LIN {X 0,Y 682.192,Z 1116.485,A -85,B 0,C 180,E1 25132.947,E2 25132.947} C_VEL
LIN {X 0,Y 681.497,Z 1132.896,A -85,B 0,C 180,E1 25130.835,E2 25130.835} C_VEL
LIN {X 0,Y 681.036,Z 1145.573,A -85,B 0,C 180,E1 25129,E2 25129} C_VEL
LIN {X 0,Y 680.643,Z 1157.899,A -85,B 0,C 180,E1 25126.991,E2 25126.991} C_VEL
LIN {X 0,Y 680.337,Z 1169.837,A -85,B 0,C 180,E1 25124.73,E2 25124.73} C_VEL
LIN {X 0,Y 680.158,Z 1178.436,A -85,B 0,C 180,E1 25122.826,E2 25122.826} C_VEL
LIN {X 0,Y 680.019,Z 1186.222,A -85,B 0,C 180,E1 25120.82,E2 25120.82} C_VEL
LIN {X 0,Y 679.964,Z 1193.353,A -85,B 0,C 180,E1 25118.541,E2 25118.541} C_VEL
LIN {X 0,Y 679.927,Z 1198.829,A -85,B 0,C 180,E1 25116.216,E2 25116.216} C_VEL
LIN {X 0,Y 679.913,Z 1202.374,A -85,B 0,C 180,E1 25114.048,E2 25114.048} C_VEL
LIN {X 0,Y 679.907,Z 1204.493,A -85,B 0,C 180,E1 25111.77,E2 25111.77} C_VEL
LIN {X 0,Y 679.891,Z 1204.872,A -85,B 0,C 180,E1 25109.495,E2 25109.495} C_VEL
LIN {X 0,Y 679.907,Z 1203.956,A -85,B 0,C 180,E1 25107.472,E2 25107.472} C_VEL
LIN {X 0,Y 679.912,Z 1201.428,A -85,B 0,C 180,E1 25105.276,E2 25105.276} C_VEL
LIN {X 0,Y 679.934,Z 1197.152,A -85,B 0,C 180,E1 25102.99,E2 25102.99} C_VEL
LIN {X 0,Y 679.978,Z 1191.385,A -85,B 0,C 180,E1 25100.777,E2 25100.777} C_VEL
LIN {X 0,Y 680.067,Z 1184.278,A -85,B 0,C 180,E1 25098.638,E2 25098.638} C_VEL
LIN {X 0,Y 680.24,Z 1173.938,A -85,B 0,C 180,E1 25096.138,E2 25096.138} C_VEL
LIN {X 0,Y 680.464,Z 1164.538,A -85,B 0,C 180,E1 25094.227,E2 25094.227} C_VEL
LIN {X 0,Y 680.75,Z 1154.23,A -85,B 0,C 180,E1 25092.388,E2 25092.388} C_VEL
LIN {X 0,Y 681.149,Z 1141.939,A -85,B 0,C 180,E1 25090.447,E2 25090.447} C_VEL
LIN {X 0,Y 681.795,Z 1125.467,A -85,B 0,C 180,E1 25088.177,E2 25088.177} C_VEL
LIN {X 0,Y 682.441,Z 1111.072,A -85,B 0,C 180,E1 25086.423,E2 25086.423} C_VEL
LIN {X 0,Y 683.271,Z 1093.72,A -85,B 0,C 180,E1 25084.518,E2 25084.518} C_VEL
LIN {X 0,Y 684.267,Z 1074.728,A -85,B 0,C 180,E1 25082.679,E2 25082.679} C_VEL
LIN {X 0,Y 685.157,Z 1057.951,A -85,B 0,C 180,E1 25081.212,E2 25081.212} C_VEL
LIN {X 0,Y 686.261,Z 1038.591,A -85,B 0,C 180,E1 25079.679,E2 25079.679} C_VEL
LIN {X 0,Y 687.621,Z 1015.177,A -85,B 0,C 180,E1 25078.043,E2 25078.043} C_VEL
LIN {X 0,Y 688.735,Z 995.445,A -85,B 0,C 180,E1 25076.818,E2 25076.818} C_VEL
LIN {X 0,Y 689.844,Z 975.494,A -85,B 0,C 180,E1 25075.709,E2 25075.709} C_VEL
LIN {X 0,Y 691.118,Z 951.69,A -85,B 0,C 180,E1 25074.54,E2 25074.54} C_VEL
LIN {X 0,Y 692.335,Z 926.424,A -85,B 0,C 180,E1 25073.487,E2 25073.487} C_VEL
LIN {X 0,Y 693.317,Z 904.137,A -85,B 0,C 180,E1 25072.695,E2 25072.695} C_VEL
LIN {X 0,Y 694.253,Z 881.059,A -85,B 0,C 180,E1 25072.001,E2 25072.001} C_VEL
LIN {X 0,Y 695.167,Z 854.051,A -85,B 0,C 180,E1 25071.355,E2 25071.355} C_VEL
LIN {X 0,Y 695.825,Z 826.957,A -85,B 0,C 180,E1 25070.881,E2 25070.881} C_VEL
LIN {X 0,Y 698.216,Z 605.17,A -85,B 0,C 180,E1 25068.081,E2 25068.081} C_VEL
LIN {X 0,Y 700.479,Z 401.113,A -85,B 0,C 180,E1 25065.437,E2 25065.437} C_VEL
LIN {X 0,Y 700.65,Z 371.915,A -85,B 0,C 180,E1 25065.038,E2 25065.038} C_VEL
LIN {X 0,Y 697.922,Z 362.234,A -85,B 0,C 180,E1 25064.675,E2 25064.675} C_VEL
LIN {X 0,Y 690.093,Z 350.368,A -85,B 0,C 180,E1 25063.818,E2 25063.818} C_VEL
LIN {X 0,Y 683.619,Z 336.797,A -85,B 0,C 180,E1 25062.172,E2 25062.172} C_VEL
LIN {X 0,Y 681.934,Z 333.218,A -85,B 0,C 180,E1 25061.729,E2 25061.729} C_VEL
LIN {X 0,Y 680.487,Z 329.763,A -85,B 0,C 180,E1 25061.314,E2 25061.314} C_VEL
LIN {X 0,Y 680.455,Z 329.473,A -85,B 0,C 180,E1 25061.171,E2 25061.171} C_VEL
LIN {X 0,Y 680.483,Z 329.469,A -85,B 0,C 180,E1 25058.108,E2 25058.108} C_VEL
LIN {X 0,Y 680.435,Z 329.466,A -85,B 0,C 180,E1 25055.482,E2 25055.482} C_VEL
LIN {X 0,Y 680.45,Z 329.467,A -85,B 0,C 180,E1 25052.936,E2 25052.936} C_VEL
LIN {X 0,Y 680.456,Z 329.462,A -85,B 0,C 180,E1 25049.78,E2 25049.78} C_VEL
LIN {X 0,Y 680.427,Z 329.462,A -85,B 0,C 180,E1 25047.249,E2 25047.249} C_VEL
LIN {X 0,Y 680.448,Z 329.464,A -85,B 0,C 180,E1 25044.666,E2 25044.666} C_VEL
LIN {X 0,Y 680.443,Z 329.453,A -85,B 0,C 180,E1 25041.542,E2 25041.542} C_VEL
LIN {X 0,Y 680.419,Z 329.47,A -85,B 0,C 180,E1 25039.04,E2 25039.04} C_VEL
LIN {X 0,Y 680.439,Z 329.451,A -85,B 0,C 180,E1 25036.476,E2 25036.476} C_VEL
LIN {X 0,Y 680.438,Z 329.466,A -85,B 0,C 180,E1 25033.339,E2 25033.339} C_VEL
LIN {X 0,Y 680.416,Z 329.454,A -85,B 0,C 180,E1 25030.842,E2 25030.842} C_VEL
LIN {X 0,Y 680.444,Z 329.47,A -85,B 0,C 180,E1 25028.28,E2 25028.28} C_VEL
LIN {X 0,Y 680.446,Z 329.459,A -85,B 0,C 180,E1 25025.143,E2 25025.143} C_VEL
LIN {X 0,Y 680.427,Z 329.468,A -85,B 0,C 180,E1 25022.611,E2 25022.611} C_VEL
LIN {X 0,Y 680.462,Z 329.448,A -85,B 0,C 180,E1 25020,E2 25020} C_VEL
LIN {X 0,Y 680.449,Z 329.464,A -85,B 0,C 180,E1 25016.883,E2 25016.883} C_VEL
LIN {X 0,Y 680.432,Z 329.449,A -85,B 0,C 180,E1 25014.35,E2 25014.35} C_VEL
LIN {X 0,Y 680.495,Z 329.469,A -85,B 0,C 180,E1 25011.636,E2 25011.636} C_VEL
LIN {X 0,Y 680.452,Z 329.458,A -85,B 0,C 180,E1 25008.644,E2 25008.644} C_VEL
LIN {X 0,Y 680.443,Z 329.466,A -85,B 0,C 180,E1 25006.141,E2 25006.141} C_VEL
LIN {X 0,Y 680.523,Z 329.45,A -85,B 0,C 180,E1 25003.263,E2 25003.263} C_VEL
LIN {X 0,Y 680.452,Z 329.455,A -85,B 0,C 180,E1 25000.336,E2 25000.336} C_VEL
LIN {X 0,Y 680.457,Z 329.465,A -85,B 0,C 180,E1 24997.778,E2 24997.778} C_VEL
LIN {X 0,Y 680.518,Z 329.449,A -85,B 0,C 180,E1 24994.78,E2 24994.78} C_VEL
LIN {X 0,Y 680.455,Z 329.464,A -85,B 0,C 180,E1 24991.951,E2 24991.951} C_VEL
LIN {X 0,Y 680.471,Z 329.465,A -85,B 0,C 180,E1 24989.482,E2 24989.482} C_VEL
LIN {X 0,Y 679.538,Z 329.59,A -85,B 0,C 180,E1 24988.834,E2 24988.834} C_VEL
LIN {X 0,Y 673.042,Z 330.4,A -85,B 0,C 180,E1 24986.969,E2 24986.969} C_VEL
LIN {X 0,Y 672.579,Z 330.454,A -85,B 0,C 180,E1 24986.544,E2 24986.544} C_VEL
LIN {X 0,Y 672.608,Z 330.615,A -85,B 0,C 180,E1 24984.551,E2 24984.551} C_VEL
LIN {X 0,Y 673.956,Z 334.1,A -85,B 0,C 180,E1 24984.124,E2 24984.124} C_VEL
LIN {X 0,Y 677.383,Z 341.291,A -85,B 0,C 180,E1 24983.233,E2 24983.233} C_VEL
LIN {X 0,Y 692.08,Z 362.695,A -85,B 0,C 180,E1 24981.619,E2 24981.619} C_VEL
LIN {X 0,Y 695.109,Z 367.708,A -85,B 0,C 180,E1 24981.292,E2 24981.292} C_VEL
LIN {X 0,Y 692.375,Z 585.7,A -85,B 0,C 180,E1 24978.44,E2 24978.44} C_VEL
LIN {X 0,Y 689.696,Z 812.863,A -85,B 0,C 180,E1 24975.554,E2 24975.554} C_VEL
LIN {X 0,Y 689.06,Z 837.442,A -85,B 0,C 180,E1 24975.148,E2 24975.148} C_VEL
LIN {X 0,Y 688.188,Z 863.617,A -85,B 0,C 180,E1 24974.567,E2 24974.567} C_VEL
LIN {X 0,Y 687.053,Z 889.758,A -85,B 0,C 180,E1 24973.816,E2 24973.816} C_VEL
LIN {X 0,Y 686.051,Z 911.255,A -85,B 0,C 180,E1 24973.069,E2 24973.069} C_VEL
LIN {X 0,Y 685.026,Z 930.752,A -85,B 0,C 180,E1 24972.289,E2 24972.289} C_VEL
LIN {X 0,Y 683.925,Z 950.165,A -85,B 0,C 180,E1 24971.409,E2 24971.409} C_VEL
LIN {X 0,Y 682.742,Z 969.945,A -85,B 0,C 180,E1 24970.398,E2 24970.398} C_VEL
LIN {X 0,Y 681.349,Z 992.918,A -85,B 0,C 180,E1 24969.075,E2 24969.075} C_VEL
LIN {X 0,Y 679.821,Z 1015.891,A -85,B 0,C 180,E1 24967.555,E2 24967.555} C_VEL
LIN {X 0,Y 678.685,Z 1034.023,A -85,B 0,C 180,E1 24966.211,E2 24966.211} C_VEL
LIN {X 0,Y 677.553,Z 1052.755,A -85,B 0,C 180,E1 24964.677,E2 24964.677} C_VEL
LIN {X 0,Y 676.24,Z 1074.005,A -85,B 0,C 180,E1 24962.719,E2 24962.719} C_VEL
LIN {X 0,Y 675.312,Z 1090.747,A -85,B 0,C 180,E1 24960.986,E2 24960.986} C_VEL
LIN {X 0,Y 674.385,Z 1108.733,A -85,B 0,C 180,E1 24958.904,E2 24958.904} C_VEL
LIN {X 0,Y 673.661,Z 1123.806,A -85,B 0,C 180,E1 24956.916,E2 24956.916} C_VEL
LIN {X 0,Y 673.147,Z 1136.6,A -85,B 0,C 180,E1 24955.029,E2 24955.029} C_VEL
LIN {X 0,Y 672.653,Z 1150.249,A -85,B 0,C 180,E1 24952.735,E2 24952.735} C_VEL
LIN {X 0,Y 672.371,Z 1160.899,A -85,B 0,C 180,E1 24950.636,E2 24950.636} C_VEL
LIN {X 0,Y 672.18,Z 1169.232,A -85,B 0,C 180,E1 24948.741,E2 24948.741} C_VEL
LIN {X 0,Y 672.043,Z 1176.964,A -85,B 0,C 180,E1 24946.687,E2 24946.687} C_VEL
LIN {X 0,Y 671.967,Z 1183.913,A -85,B 0,C 180,E1 24944.388,E2 24944.388} C_VEL
LIN {X 0,Y 671.924,Z 1189.086,A -85,B 0,C 180,E1 24942.111,E2 24942.111} C_VEL
LIN {X 0,Y 671.91,Z 1192.514,A -85,B 0,C 180,E1 24939.94,E2 24939.94} C_VEL
LIN {X 0,Y 671.907,Z 1194.57,A -85,B 0,C 180,E1 24937.61,E2 24937.61} C_VEL
LIN {X 0,Y 671.898,Z 1194.855,A -85,B 0,C 180,E1 24935.379,E2 24935.379} C_VEL
LIN {X 0,Y 671.907,Z 1193.966,A -85,B 0,C 180,E1 24933.412,E2 24933.412} C_VEL
LIN {X 0,Y 671.914,Z 1191.456,A -85,B 0,C 180,E1 24931.193,E2 24931.193} C_VEL
LIN {X 0,Y 671.941,Z 1187.221,A -85,B 0,C 180,E1 24928.891,E2 24928.891} C_VEL
LIN {X 0,Y 671.989,Z 1181.533,A -85,B 0,C 180,E1 24926.673,E2 24926.673} C_VEL
LIN {X 0,Y 672.093,Z 1174.22,A -85,B 0,C 180,E1 24924.44,E2 24924.44} C_VEL
LIN {X 0,Y 672.267,Z 1164.112,A -85,B 0,C 180,E1 24921.963,E2 24921.963} C_VEL
LIN {X 0,Y 672.539,Z 1154.496,A -85,B 0,C 180,E1 24919.982,E2 24919.982} C_VEL
LIN {X 0,Y 672.864,Z 1144.443,A -85,B 0,C 180,E1 24918.166,E2 24918.166} C_VEL
LIN {X 0,Y 673.321,Z 1131.955,A -85,B 0,C 180,E1 24916.167,E2 24916.167} C_VEL
LIN {X 0,Y 674.037,Z 1115.678,A -85,B 0,C 180,E1 24913.895,E2 24913.895} C_VEL
LIN {X 0,Y 674.762,Z 1100.696,A -85,B 0,C 180,E1 24912.048,E2 24912.048} C_VEL
LIN {X 0,Y 675.765,Z 1083.129,A -85,B 0,C 180,E1 24910.104,E2 24910.104} C_VEL
LIN {X 0,Y 676.829,Z 1063.955,A -85,B 0,C 180,E1 24908.235,E2 24908.235} C_VEL
LIN {X 0,Y 677.883,Z 1046.646,A -85,B 0,C 180,E1 24906.715,E2 24906.715} C_VEL
LIN {X 0,Y 679.31,Z 1025.059,A -85,B 0,C 180,E1 24905.011,E2 24905.011} C_VEL
LIN {X 0,Y 680.632,Z 1003.591,A -85,B 0,C 180,E1 24903.522,E2 24903.522} C_VEL
LIN {X 0,Y 681.817,Z 984.728,A -85,B 0,C 180,E1 24902.347,E2 24902.347} C_VEL
LIN {X 0,Y 683.115,Z 963.487,A -85,B 0,C 180,E1 24901.165,E2 24901.165} C_VEL
LIN {X 0,Y 684.679,Z 937.06,A -85,B 0,C 180,E1 24899.892,E2 24899.892} C_VEL
LIN {X 0,Y 685.803,Z 915.856,A -85,B 0,C 180,E1 24899.015,E2 24899.015} C_VEL
LIN {X 0,Y 686.762,Z 895.765,A -85,B 0,C 180,E1 24898.292,E2 24898.292} C_VEL
LIN {X 0,Y 687.782,Z 873.499,A -85,B 0,C 180,E1 24897.609,E2 24897.609} C_VEL
LIN {X 0,Y 688.802,Z 846.613,A -85,B 0,C 180,E1 24896.945,E2 24896.945} C_VEL
LIN {X 0,Y 689.546,Z 819.591,A -85,B 0,C 180,E1 24896.454,E2 24896.454} C_VEL
LIN {X 0,Y 690.716,Z 728.303,A -85,B 0,C 180,E1 24895.287,E2 24895.287} C_VEL
LIN {X 0,Y 693.173,Z 517.537,A -85,B 0,C 180,E1 24892.586,E2 24892.586} C_VEL
LIN {X 0,Y 695.013,Z 367.196,A -85,B 0,C 180,E1 24890.603,E2 24890.603} C_VEL
LIN {X 0,Y 681.213,Z 346.68,A -85,B 0,C 180,E1 24889.106,E2 24889.106} C_VEL
LIN {X 0,Y 676.997,Z 340.608,A -85,B 0,C 180,E1 24888.616,E2 24888.616} C_VEL
LIN {X 0,Y 673.889,Z 333.927,A -85,B 0,C 180,E1 24887.766,E2 24887.766} C_VEL
LIN {X 0,Y 672.576,Z 330.451,A -85,B 0,C 180,E1 24887.319,E2 24887.319} C_VEL
LIN {X 0,Y 672.555,Z 330.455,A -85,B 0,C 180,E1 24884.349,E2 24884.349} C_VEL
LIN {X 0,Y 672.579,Z 330.449,A -85,B 0,C 180,E1 24881.345,E2 24881.345} C_VEL
LIN {X 0,Y 672.555,Z 330.453,A -85,B 0,C 180,E1 24878.419,E2 24878.419} C_VEL
LIN {X 0,Y 672.585,Z 330.446,A -85,B 0,C 180,E1 24875.436,E2 24875.436} C_VEL
LIN {X 0,Y 672.552,Z 330.456,A -85,B 0,C 180,E1 24872.359,E2 24872.359} C_VEL
LIN {X 0,Y 672.579,Z 330.447,A -85,B 0,C 180,E1 24869.38,E2 24869.38} C_VEL
LIN {X 0,Y 672.548,Z 330.431,A -85,B 0,C 180,E1 24866.298,E2 24866.298} C_VEL
LIN {X 0,Y 672.559,Z 330.449,A -85,B 0,C 180,E1 24863.388,E2 24863.388} C_VEL
LIN {X 0,Y 672.549,Z 330.429,A -85,B 0,C 180,E1 24860.264,E2 24860.264} C_VEL
LIN {X 0,Y 672.536,Z 330.451,A -85,B 0,C 180,E1 24857.477,E2 24857.477} C_VEL
LIN {X 0,Y 672.572,Z 330.425,A -85,B 0,C 180,E1 24854.375,E2 24854.375} C_VEL
LIN {X 0,Y 672.522,Z 330.45,A -85,B 0,C 180,E1 24851.543,E2 24851.543} C_VEL
LIN {X 0,Y 672.588,Z 330.446,A -85,B 0,C 180,E1 24848.636,E2 24848.636} C_VEL
LIN {X 0,Y 672.518,Z 330.449,A -85,B 0,C 180,E1 24845.717,E2 24845.717} C_VEL
LIN {X 0,Y 672.525,Z 330.453,A -85,B 0,C 180,E1 24843.068,E2 24843.068} C_VEL
LIN {X 0,Y 672.541,Z 330.456,A -85,B 0,C 180,E1 24839.915,E2 24839.915} C_VEL
LIN {X 0,Y 672.504,Z 330.453,A -85,B 0,C 180,E1 24837.273,E2 24837.273} C_VEL
LIN {X 0,Y 672.564,Z 330.448,A -85,B 0,C 180,E1 24834.455,E2 24834.455} C_VEL
LIN {X 0,Y 672.503,Z 330.451,A -85,B 0,C 180,E1 24831.449,E2 24831.449} C_VEL
LIN {X 0,Y 672.498,Z 330.456,A -85,B 0,C 180,E1 24828.901,E2 24828.901} C_VEL
LIN {X 0,Y 672.576,Z 330.427,A -85,B 0,C 180,E1 24825.976,E2 24825.976} C_VEL
LIN {X 0,Y 672.488,Z 330.458,A -85,B 0,C 180,E1 24823.146,E2 24823.146} C_VEL
LIN {X 0,Y 672.49,Z 330.439,A -85,B 0,C 180,E1 24820.636,E2 24820.636} C_VEL
LIN {X 0,Y 672.539,Z 330.458,A -85,B 0,C 180,E1 24817.629,E2 24817.629} C_VEL
LIN {X 0,Y 672.477,Z 330.434,A -85,B 0,C 180,E1 24814.89,E2 24814.89} C_VEL
LIN {X 0,Y 672.507,Z 330.458,A -85,B 0,C 180,E1 24812.266,E2 24812.266} C_VEL
LIN {X 0,Y 672.508,Z 330.453,A -85,B 0,C 180,E1 24809.139,E2 24809.139} C_VEL
LIN {X 0,Y 672.491,Z 330.46,A -85,B 0,C 180,E1 24806.624,E2 24806.624} C_VEL
LIN {X 0,Y 672.537,Z 330.459,A -85,B 0,C 180,E1 24803.931,E2 24803.931} C_VEL
LIN {X 0,Y 672.515,Z 330.464,A -85,B 0,C 180,E1 24800.905,E2 24800.905} C_VEL
LIN {X 0,Y 672.607,Z 330.647,A -85,B 0,C 180,E1 24799.373,E2 24799.373} C_VEL
LIN {X 0,Y 673.722,Z 333.767,A -85,B 0,C 180,E1 24799.005,E2 24799.005} C_VEL
LIN {X 0,Y 674.749,Z 335.752,A -85,B 0,C 180,E1 24798.743,E2 24798.743} C_VEL
LIN {X 0,Y 680.465,Z 347.723,A -85,B 0,C 180,E1 24797.244,E2 24797.244} C_VEL
LIN {X 0,Y 682.244,Z 351.282,A -85,B 0,C 180,E1 24796.838,E2 24796.838} C_VEL
LIN {X 0,Y 693.378,Z 368.095,A -85,B 0,C 180,E1 24795.621,E2 24795.621} C_VEL
LIN {X 0,Y 695.107,Z 375.541,A -85,B 0,C 180,E1 24795.368,E2 24795.368} C_VEL
LIN {X 0,Y 692.464,Z 587.805,A -85,B 0,C 180,E1 24792.587,E2 24792.587} C_VEL
LIN {X 0,Y 689.907,Z 810.343,A -85,B 0,C 180,E1 24789.763,E2 24789.763} C_VEL
LIN {X 0,Y 689.271,Z 840.613,A -85,B 0,C 180,E1 24789.32,E2 24789.32} C_VEL
LIN {X 0,Y 688.468,Z 865.299,A -85,B 0,C 180,E1 24788.812,E2 24788.812} C_VEL
LIN {X 0,Y 687.48,Z 890.926,A -85,B 0,C 180,E1 24788.136,E2 24788.136} C_VEL
LIN {X 0,Y 686.225,Z 918.026,A -85,B 0,C 180,E1 24787.235,E2 24787.235} C_VEL
LIN {X 0,Y 685.097,Z 939.47,A -85,B 0,C 180,E1 24786.39,E2 24786.39} C_VEL
LIN {X 0,Y 683.956,Z 959.707,A -85,B 0,C 180,E1 24785.477,E2 24785.477} C_VEL
LIN {X 0,Y 682.726,Z 980.321,A -85,B 0,C 180,E1 24784.424,E2 24784.424} C_VEL
LIN {X 0,Y 681.2,Z 1004.925,A -85,B 0,C 180,E1 24782.995,E2 24782.995} C_VEL
LIN {X 0,Y 679.764,Z 1026.908,A -85,B 0,C 180,E1 24781.528,E2 24781.528} C_VEL
LIN {X 0,Y 678.598,Z 1045.712,A -85,B 0,C 180,E1 24780.125,E2 24780.125} C_VEL
LIN {X 0,Y 677.318,Z 1066.768,A -85,B 0,C 180,E1 24778.376,E2 24778.376} C_VEL
LIN {X 0,Y 676.139,Z 1085.449,A -85,B 0,C 180,E1 24776.621,E2 24776.621} C_VEL
LIN {X 0,Y 675.284,Z 1101.386,A -85,B 0,C 180,E1 24774.961,E2 24774.961} C_VEL
LIN {X 0,Y 674.296,Z 1120.132,A -85,B 0,C 180,E1 24772.77,E2 24772.77} C_VEL
LIN {X 0,Y 673.636,Z 1134.458,A -85,B 0,C 180,E1 24770.869,E2 24770.869} C_VEL
LIN {X 0,Y 673.123,Z 1147.165,A -85,B 0,C 180,E1 24768.985,E2 24768.985} C_VEL
LIN {X 0,Y 672.64,Z 1160.81,A -85,B 0,C 180,E1 24766.672,E2 24766.672} C_VEL
LIN {X 0,Y 672.363,Z 1171.07,A -85,B 0,C 180,E1 24764.644,E2 24764.644} C_VEL
LIN {X 0,Y 672.177,Z 1179.152,A -85,B 0,C 180,E1 24762.806,E2 24762.806} C_VEL
LIN {X 0,Y 672.03,Z 1186.718,A -85,B 0,C 180,E1 24760.805,E2 24760.805} C_VEL
LIN {X 0,Y 671.969,Z 1193.594,A -85,B 0,C 180,E1 24758.558,E2 24758.558} C_VEL
LIN {X 0,Y 671.929,Z 1198.936,A -85,B 0,C 180,E1 24756.237,E2 24756.237} C_VEL
LIN {X 0,Y 671.915,Z 1202.371,A -85,B 0,C 180,E1 24754.096,E2 24754.096} C_VEL
LIN {X 0,Y 671.907,Z 1204.494,A -85,B 0,C 180,E1 24751.791,E2 24751.791} C_VEL
LIN {X 0,Y 671.891,Z 1204.872,A -85,B 0,C 180,E1 24749.489,E2 24749.489} C_VEL
LIN {X 0,Y 671.907,Z 1203.953,A -85,B 0,C 180,E1 24747.442,E2 24747.442} C_VEL
LIN {X 0,Y 671.914,Z 1201.428,A -85,B 0,C 180,E1 24745.22,E2 24745.22} C_VEL
LIN {X 0,Y 671.941,Z 1197.152,A -85,B 0,C 180,E1 24742.906,E2 24742.906} C_VEL
LIN {X 0,Y 671.991,Z 1191.382,A -85,B 0,C 180,E1 24740.667,E2 24740.667} C_VEL
LIN {X 0,Y 672.091,Z 1184.278,A -85,B 0,C 180,E1 24738.501,E2 24738.501} C_VEL
LIN {X 0,Y 672.286,Z 1173.937,A -85,B 0,C 180,E1 24735.971,E2 24735.971} C_VEL
LIN {X 0,Y 672.534,Z 1164.54,A -85,B 0,C 180,E1 24734.036,E2 24734.036} C_VEL
LIN {X 0,Y 672.866,Z 1154.232,A -85,B 0,C 180,E1 24732.175,E2 24732.175} C_VEL
LIN {X 0,Y 673.319,Z 1141.941,A -85,B 0,C 180,E1 24730.21,E2 24730.21} C_VEL
LIN {X 0,Y 674.025,Z 1125.809,A -85,B 0,C 180,E1 24727.957,E2 24727.957} C_VEL
LIN {X 0,Y 674.751,Z 1111.073,A -85,B 0,C 180,E1 24726.138,E2 24726.138} C_VEL
LIN {X 0,Y 675.713,Z 1093.721,A -85,B 0,C 180,E1 24724.212,E2 24724.212} C_VEL
LIN {X 0,Y 676.818,Z 1074.326,A -85,B 0,C 180,E1 24722.315,E2 24722.315} C_VEL
LIN {X 0,Y 677.817,Z 1057.658,A -85,B 0,C 180,E1 24720.845,E2 24720.845} C_VEL
LIN {X 0,Y 679.09,Z 1037.98,A -85,B 0,C 180,E1 24719.276,E2 24719.276} C_VEL
LIN {X 0,Y 680.589,Z 1014.452,A -85,B 0,C 180,E1 24717.623,E2 24717.623} C_VEL
LIN {X 0,Y 681.824,Z 994.646,A -85,B 0,C 180,E1 24716.387,E2 24716.387} C_VEL
LIN {X 0,Y 683.131,Z 973.165,A -85,B 0,C 180,E1 24715.192,E2 24715.192} C_VEL
LIN {X 0,Y 684.732,Z 946.223,A -85,B 0,C 180,E1 24713.9,E2 24713.9} C_VEL
LIN {X 0,Y 685.855,Z 925.015,A -85,B 0,C 180,E1 24713.027,E2 24713.027} C_VEL
LIN {X 0,Y 686.853,Z 904.064,A -85,B 0,C 180,E1 24712.28,E2 24712.28} C_VEL
LIN {X 0,Y 687.876,Z 880.997,A -85,B 0,C 180,E1 24711.584,E2 24711.584} C_VEL
LIN {X 0,Y 688.888,Z 854.053,A -85,B 0,C 180,E1 24710.936,E2 24710.936} C_VEL
LIN {X 0,Y 689.604,Z 827.138,A -85,B 0,C 180,E1 24710.463,E2 24710.463} C_VEL
LIN {X 0,Y 692.229,Z 607.714,A -85,B 0,C 180,E1 24707.669,E2 24707.669} C_VEL
LIN {X 0,Y 694.743,Z 403.368,A -85,B 0,C 180,E1 24705.001,E2 24705.001} C_VEL
LIN {X 0,Y 694.947,Z 374.179,A -85,B 0,C 180,E1 24704.599,E2 24704.599} C_VEL
LIN {X 0,Y 692.936,Z 367.154,A -85,B 0,C 180,E1 24704.328,E2 24704.328} C_VEL
LIN {X 0,Y 683.819,Z 353.781,A -85,B 0,C 180,E1 24703.34,E2 24703.34} C_VEL
LIN {X 0,Y 681.644,Z 350.368,A -85,B 0,C 180,E1 24703.073,E2 24703.073} C_VEL
LIN {X 0,Y 676.08,Z 338.51,A -85,B 0,C 180,E1 24701.61,E2 24701.61} C_VEL
LIN {X 0,Y 673.717,Z 333.758,A -85,B 0,C 180,E1 24700.995,E2 24700.995} C_VEL
LIN {X 0,Y 672.584,Z 330.454,A -85,B 0,C 180,E1 24700.598,E2 24700.598} C_VEL
LIN {X 0,Y 672.504,Z 330.459,A -85,B 0,C 180,E1 24697.668,E2 24697.668} C_VEL
LIN {X 0,Y 672.503,Z 330.454,A -85,B 0,C 180,E1 24695.128,E2 24695.128} C_VEL
LIN {X 0,Y 672.566,Z 330.451,A -85,B 0,C 180,E1 24692.157,E2 24692.157} C_VEL
LIN {X 0,Y 672.493,Z 330.456,A -85,B 0,C 180,E1 24689.384,E2 24689.384} C_VEL
LIN {X 0,Y 672.492,Z 330.449,A -85,B 0,C 180,E1 24686.968,E2 24686.968} C_VEL
LIN {X 0,Y 672.57,Z 330.457,A -85,B 0,C 180,E1 24684.038,E2 24684.038} C_VEL
LIN {X 0,Y 672.485,Z 330.444,A -85,B 0,C 180,E1 24681.272,E2 24681.272} C_VEL
LIN {X 0,Y 672.484,Z 330.459,A -85,B 0,C 180,E1 24678.823,E2 24678.823} C_VEL
LIN {X 0,Y 672.565,Z 330.436,A -85,B 0,C 180,E1 24675.875,E2 24675.875} C_VEL
LIN {X 0,Y 672.481,Z 330.455,A -85,B 0,C 180,E1 24673.062,E2 24673.062} C_VEL
LIN {X 0,Y 672.486,Z 330.442,A -85,B 0,C 180,E1 24670.538,E2 24670.538} C_VEL
LIN {X 0,Y 672.548,Z 330.447,A -85,B 0,C 180,E1 24667.518,E2 24667.518} C_VEL
LIN {X 0,Y 672.486,Z 330.449,A -85,B 0,C 180,E1 24664.776,E2 24664.776} C_VEL
LIN {X 0,Y 672.506,Z 330.458,A -85,B 0,C 180,E1 24662.215,E2 24662.215} C_VEL
LIN {X 0,Y 672.52,Z 330.452,A -85,B 0,C 180,E1 24659.063,E2 24659.063} C_VEL
LIN {X 0,Y 672.494,Z 330.454,A -85,B 0,C 180,E1 24656.42,E2 24656.42} C_VEL
LIN {X 0,Y 672.566,Z 330.439,A -85,B 0,C 180,E1 24653.598,E2 24653.598} C_VEL
LIN {X 0,Y 672.505,Z 330.447,A -85,B 0,C 180,E1 24650.587,E2 24650.587} C_VEL
LIN {X 0,Y 672.511,Z 330.448,A -85,B 0,C 180,E1 24647.986,E2 24647.986} C_VEL
LIN {X 0,Y 672.569,Z 330.43,A -85,B 0,C 180,E1 24645.008,E2 24645.008} C_VEL
LIN {X 0,Y 672.508,Z 330.455,A -85,B 0,C 180,E1 24642.165,E2 24642.165} C_VEL
LIN {X 0,Y 672.562,Z 330.435,A -85,B 0,C 180,E1 24639.369,E2 24639.369} C_VEL
LIN {X 0,Y 672.524,Z 330.448,A -85,B 0,C 180,E1 24636.324,E2 24636.324} C_VEL
LIN {X 0,Y 672.522,Z 330.454,A -85,B 0,C 180,E1 24633.701,E2 24633.701} C_VEL
LIN {X 0,Y 672.588,Z 330.446,A -85,B 0,C 180,E1 24630.718,E2 24630.718} C_VEL
LIN {X 0,Y 672.522,Z 330.456,A -85,B 0,C 180,E1 24627.841,E2 24627.841} C_VEL
LIN {X 0,Y 672.579,Z 330.454,A -85,B 0,C 180,E1 24626.544,E2 24626.544} C_VEL
LIN {X 0,Y 671.671,Z 330.679,A -85,B 0,C 180,E1 24626.089,E2 24626.089} C_VEL
LIN {X 0,Y 668.299,Z 332.282,A -85,B 0,C 180,E1 24625.356,E2 24625.356} C_VEL
LIN {X 0,Y 666.743,Z 334.518,A -85,B 0,C 180,E1 24624.891,E2 24624.891} C_VEL
LIN {X 0,Y 666.809,Z 336.494,A -85,B 0,C 180,E1 24624.619,E2 24624.619} C_VEL
LIN {X 0,Y 669.158,Z 341.54,A -85,B 0,C 180,E1 24623.999,E2 24623.999} C_VEL
LIN {X 0,Y 681.76,Z 359.579,A -85,B 0,C 180,E1 24622.561,E2 24622.561} C_VEL
LIN {X 0,Y 689.425,Z 371.303,A -85,B 0,C 180,E1 24621.719,E2 24621.719} C_VEL
LIN {X 0,Y 686.412,Z 590.021,A -85,B 0,C 180,E1 24618.837,E2 24618.837} C_VEL
LIN {X 0,Y 683.502,Z 813.654,A -85,B 0,C 180,E1 24615.971,E2 24615.971} C_VEL
LIN {X 0,Y 682.82,Z 837.703,A -85,B 0,C 180,E1 24615.57,E2 24615.57} C_VEL
LIN {X 0,Y 681.871,Z 863.883,A -85,B 0,C 180,E1 24614.985,E2 24614.985} C_VEL
LIN {X 0,Y 680.67,Z 889.429,A -85,B 0,C 180,E1 24614.247,E2 24614.247} C_VEL
LIN {X 0,Y 679.567,Z 910.882,A -85,B 0,C 180,E1 24613.499,E2 24613.499} C_VEL
LIN {X 0,Y 678.47,Z 929.901,A -85,B 0,C 180,E1 24612.738,E2 24612.738} C_VEL
LIN {X 0,Y 677.219,Z 950.032,A -85,B 0,C 180,E1 24611.821,E2 24611.821} C_VEL
LIN {X 0,Y 675.915,Z 969.984,A -85,B 0,C 180,E1 24610.794,E2 24610.794} C_VEL
LIN {X 0,Y 674.346,Z 993.619,A -85,B 0,C 180,E1 24609.419,E2 24609.419} C_VEL
LIN {X 0,Y 672.654,Z 1016.598,A -85,B 0,C 180,E1 24607.877,E2 24607.877} C_VEL
LIN {X 0,Y 671.391,Z 1034.83,A -85,B 0,C 180,E1 24606.509,E2 24606.509} C_VEL
LIN {X 0,Y 670.071,Z 1054.857,A -85,B 0,C 180,E1 24604.843,E2 24604.843} C_VEL
LIN {X 0,Y 668.706,Z 1074.695,A -85,B 0,C 180,E1 24602.974,E2 24602.974} C_VEL
LIN {X 0,Y 667.715,Z 1090.61,A -85,B 0,C 180,E1 24601.306,E2 24601.306} C_VEL
LIN {X 0,Y 666.688,Z 1108.577,A -85,B 0,C 180,E1 24599.205,E2 24599.205} C_VEL
LIN {X 0,Y 665.872,Z 1123.898,A -85,B 0,C 180,E1 24597.16,E2 24597.16} C_VEL
LIN {X 0,Y 665.303,Z 1136.579,A -85,B 0,C 180,E1 24595.265,E2 24595.265} C_VEL
LIN {X 0,Y 664.771,Z 1149.955,A -85,B 0,C 180,E1 24592.998,E2 24592.998} C_VEL
LIN {X 0,Y 664.427,Z 1160.963,A -85,B 0,C 180,E1 24590.802,E2 24590.802} C_VEL
LIN {X 0,Y 664.213,Z 1169.289,A -85,B 0,C 180,E1 24588.883,E2 24588.883} C_VEL
LIN {X 0,Y 664.057,Z 1177.011,A -85,B 0,C 180,E1 24586.803,E2 24586.803} C_VEL
LIN {X 0,Y 663.975,Z 1183.982,A -85,B 0,C 180,E1 24584.463,E2 24584.463} C_VEL
LIN {X 0,Y 663.926,Z 1189.11,A -85,B 0,C 180,E1 24582.171,E2 24582.171} C_VEL
LIN {X 0,Y 663.91,Z 1192.563,A -85,B 0,C 180,E1 24579.946,E2 24579.946} C_VEL
LIN {X 0,Y 663.907,Z 1194.573,A -85,B 0,C 180,E1 24577.616,E2 24577.616} C_VEL
LIN {X 0,Y 663.899,Z 1194.851,A -85,B 0,C 180,E1 24575.358,E2 24575.358} C_VEL
LIN {X 0,Y 663.907,Z 1193.952,A -85,B 0,C 180,E1 24573.367,E2 24573.367} C_VEL
LIN {X 0,Y 663.917,Z 1191.435,A -85,B 0,C 180,E1 24571.121,E2 24571.121} C_VEL
LIN {X 0,Y 663.945,Z 1187.189,A -85,B 0,C 180,E1 24568.792,E2 24568.792} C_VEL
LIN {X 0,Y 663.999,Z 1181.49,A -85,B 0,C 180,E1 24566.546,E2 24566.546} C_VEL
LIN {X 0,Y 664.114,Z 1174.211,A -85,B 0,C 180,E1 24564.297,E2 24564.297} C_VEL
LIN {X 0,Y 664.324,Z 1164.051,A -85,B 0,C 180,E1 24561.779,E2 24561.779} C_VEL
LIN {X 0,Y 664.616,Z 1154.432,A -85,B 0,C 180,E1 24559.774,E2 24559.774} C_VEL
LIN {X 0,Y 664.986,Z 1143.865,A -85,B 0,C 180,E1 24557.848,E2 24557.848} C_VEL
LIN {X 0,Y 665.595,Z 1130.176,A -85,B 0,C 180,E1 24555.648,E2 24555.648} C_VEL
LIN {X 0,Y 666.35,Z 1114.779,A -85,B 0,C 180,E1 24553.507,E2 24553.507} C_VEL
LIN {X 0,Y 667.141,Z 1099.849,A -85,B 0,C 180,E1 24551.655,E2 24551.655} C_VEL
LIN {X 0,Y 668.313,Z 1081.252,A -85,B 0,C 180,E1 24549.598,E2 24549.598} C_VEL
LIN {X 0,Y 669.44,Z 1063.177,A -85,B 0,C 180,E1 24547.827,E2 24547.827} C_VEL
LIN {X 0,Y 670.682,Z 1045.42,A -85,B 0,C 180,E1 24546.261,E2 24546.261} C_VEL
LIN {X 0,Y 672.3,Z 1022.368,A -85,B 0,C 180,E1 24544.45,E2 24544.45} C_VEL
LIN {X 0,Y 673.639,Z 1002.717,A -85,B 0,C 180,E1 24543.082,E2 24543.082} C_VEL
LIN {X 0,Y 675.004,Z 982.947,A -85,B 0,C 180,E1 24541.849,E2 24541.849} C_VEL
LIN {X 0,Y 676.732,Z 958.249,A -85,B 0,C 180,E1 24540.49,E2 24540.49} C_VEL
LIN {X 0,Y 678.195,Z 934.629,A -85,B 0,C 180,E1 24539.377,E2 24539.377} C_VEL
LIN {X 0,Y 679.291,Z 915.742,A -85,B 0,C 180,E1 24538.596,E2 24538.596} C_VEL
LIN {X 0,Y 680.347,Z 895.338,A -85,B 0,C 180,E1 24537.858,E2 24537.858} C_VEL
LIN {X 0,Y 681.452,Z 873.122,A -85,B 0,C 180,E1 24537.175,E2 24537.175} C_VEL
LIN {X 0,Y 682.568,Z 846.2,A -85,B 0,C 180,E1 24536.509,E2 24536.509} C_VEL
LIN {X 0,Y 683.37,Z 819.214,A -85,B 0,C 180,E1 24536.02,E2 24536.02} C_VEL
LIN {X 0,Y 684.764,Z 718.371,A -85,B 0,C 180,E1 24534.722,E2 24534.722} C_VEL
LIN {X 0,Y 687.447,Z 510.327,A -85,B 0,C 180,E1 24532.031,E2 24532.031} C_VEL
LIN {X 0,Y 689.298,Z 370.726,A -85,B 0,C 180,E1 24530.172,E2 24530.172} C_VEL
LIN {X 0,Y 673.884,Z 348.149,A -85,B 0,C 180,E1 24528.46,E2 24528.46} C_VEL
LIN {X 0,Y 668.725,Z 340.57,A -85,B 0,C 180,E1 24527.829,E2 24527.829} C_VEL
LIN {X 0,Y 666.082,Z 335.117,A -85,B 0,C 180,E1 24527.102,E2 24527.102} C_VEL
LIN {X 0,Y 664.633,Z 331.51,A -85,B 0,C 180,E1 24526.642,E2 24526.642} C_VEL
LIN {X 0,Y 664.644,Z 331.438,A -85,B 0,C 180,E1 24523.552,E2 24523.552} C_VEL
LIN {X 0,Y 664.621,Z 331.445,A -85,B 0,C 180,E1 24520.536,E2 24520.536} C_VEL
LIN {X 0,Y 664.646,Z 331.434,A -85,B 0,C 180,E1 24517.538,E2 24517.538} C_VEL
LIN {X 0,Y 664.62,Z 331.445,A -85,B 0,C 180,E1 24514.449,E2 24514.449} C_VEL
LIN {X 0,Y 664.64,Z 331.438,A -85,B 0,C 180,E1 24511.462,E2 24511.462} C_VEL
LIN {X 0,Y 664.611,Z 331.435,A -85,B 0,C 180,E1 24508.289,E2 24508.289} C_VEL
LIN {X 0,Y 664.635,Z 331.421,A -85,B 0,C 180,E1 24505.292,E2 24505.292} C_VEL
LIN {X 0,Y 664.604,Z 331.433,A -85,B 0,C 180,E1 24502.187,E2 24502.187} C_VEL
LIN {X 0,Y 664.61,Z 331.42,A -85,B 0,C 180,E1 24499.329,E2 24499.329} C_VEL
LIN {X 0,Y 664.609,Z 331.437,A -85,B 0,C 180,E1 24496.161,E2 24496.161} C_VEL
LIN {X 0,Y 664.588,Z 331.413,A -85,B 0,C 180,E1 24493.397,E2 24493.397} C_VEL
LIN {X 0,Y 664.632,Z 331.444,A -85,B 0,C 180,E1 24490.301,E2 24490.301} C_VEL
LIN {X 0,Y 664.578,Z 331.442,A -85,B 0,C 180,E1 24487.482,E2 24487.482} C_VEL
LIN {X 0,Y 664.646,Z 331.433,A -85,B 0,C 180,E1 24484.573,E2 24484.573} C_VEL
LIN {X 0,Y 664.576,Z 331.439,A -85,B 0,C 180,E1 24481.638,E2 24481.638} C_VEL
LIN {X 0,Y 664.576,Z 331.442,A -85,B 0,C 180,E1 24479.052,E2 24479.052} C_VEL
LIN {X 0,Y 664.622,Z 331.443,A -85,B 0,C 180,E1 24476.032,E2 24476.032} C_VEL
LIN {X 0,Y 664.56,Z 331.445,A -85,B 0,C 180,E1 24473.225,E2 24473.225} C_VEL
LIN {X 0,Y 664.592,Z 331.438,A -85,B 0,C 180,E1 24470.561,E2 24470.561} C_VEL
LIN {X 0,Y 664.567,Z 331.426,A -85,B 0,C 180,E1 24467.487,E2 24467.487} C_VEL
LIN {X 0,Y 664.549,Z 331.437,A -85,B 0,C 180,E1 24465.001,E2 24465.001} C_VEL
LIN {X 0,Y 664.602,Z 331.443,A -85,B 0,C 180,E1 24462.238,E2 24462.238} C_VEL
LIN {X 0,Y 664.55,Z 331.438,A -85,B 0,C 180,E1 24459.201,E2 24459.201} C_VEL
LIN {X 0,Y 664.539,Z 331.447,A -85,B 0,C 180,E1 24456.783,E2 24456.783} C_VEL
LIN {X 0,Y 664.616,Z 331.419,A -85,B 0,C 180,E1 24453.917,E2 24453.917} C_VEL
LIN {X 0,Y 664.549,Z 331.445,A -85,B 0,C 180,E1 24450.947,E2 24450.947} C_VEL
LIN {X 0,Y 664.55,Z 331.442,A -85,B 0,C 180,E1 24448.527,E2 24448.527} C_VEL
LIN {X 0,Y 664.636,Z 331.445,A -85,B 0,C 180,E1 24445.656,E2 24445.656} C_VEL
LIN {X 0,Y 664.561,Z 331.45,A -85,B 0,C 180,E1 24442.742,E2 24442.742} C_VEL
LIN {X 0,Y 664.566,Z 331.455,A -85,B 0,C 180,E1 24440.249,E2 24440.249} C_VEL
LIN {X 0,Y 664.609,Z 331.683,A -85,B 0,C 180,E1 24440.084,E2 24440.084} C_VEL
LIN {X 0,Y 665.934,Z 334.932,A -85,B 0,C 180,E1 24439.673,E2 24439.673} C_VEL
LIN {X 0,Y 666.941,Z 336.884,A -85,B 0,C 180,E1 24439.408,E2 24439.408} C_VEL
LIN {X 0,Y 673.766,Z 351.136,A -85,B 0,C 180,E1 24437.614,E2 24437.614} C_VEL
LIN {X 0,Y 686.84,Z 370.214,A -85,B 0,C 180,E1 24436.15,E2 24436.15} C_VEL
LIN {X 0,Y 688.483,Z 373.277,A -85,B 0,C 180,E1 24435.963,E2 24435.963} C_VEL
LIN {X 0,Y 689.447,Z 377.743,A -85,B 0,C 180,E1 24435.814,E2 24435.814} C_VEL
LIN {X 0,Y 686.549,Z 589.284,A -85,B 0,C 180,E1 24433.022,E2 24433.022} C_VEL
LIN {X 0,Y 683.733,Z 811.997,A -85,B 0,C 180,E1 24430.173,E2 24430.173} C_VEL
LIN {X 0,Y 683.038,Z 841.238,A -85,B 0,C 180,E1 24429.736,E2 24429.736} C_VEL
LIN {X 0,Y 682.185,Z 865.409,A -85,B 0,C 180,E1 24429.235,E2 24429.235} C_VEL
LIN {X 0,Y 681.1,Z 891.03,A -85,B 0,C 180,E1 24428.556,E2 24428.556} C_VEL
LIN {X 0,Y 679.738,Z 917.896,A -85,B 0,C 180,E1 24427.657,E2 24427.657} C_VEL
LIN {X 0,Y 678.493,Z 939.466,A -85,B 0,C 180,E1 24426.802,E2 24426.802} C_VEL
LIN {X 0,Y 677.244,Z 959.704,A -85,B 0,C 180,E1 24425.883,E2 24425.883} C_VEL
LIN {X 0,Y 675.887,Z 980.552,A -85,B 0,C 180,E1 24424.809,E2 24424.809} C_VEL
LIN {X 0,Y 674.237,Z 1004.923,A -85,B 0,C 180,E1 24423.38,E2 24423.38} C_VEL
LIN {X 0,Y 672.654,Z 1026.643,A -85,B 0,C 180,E1 24421.92,E2 24421.92} C_VEL
LIN {X 0,Y 671.372,Z 1045.259,A -85,B 0,C 180,E1 24420.521,E2 24420.521} C_VEL
LIN {X 0,Y 669.982,Z 1066.194,A -85,B 0,C 180,E1 24418.77,E2 24418.77} C_VEL
LIN {X 0,Y 668.655,Z 1085.188,A -85,B 0,C 180,E1 24416.97,E2 24416.97} C_VEL
LIN {X 0,Y 667.706,Z 1100.539,A -85,B 0,C 180,E1 24415.359,E2 24415.359} C_VEL
LIN {X 0,Y 666.721,Z 1118.002,A -85,B 0,C 180,E1 24413.324,E2 24413.324} C_VEL
LIN {X 0,Y 665.878,Z 1133.816,A -85,B 0,C 180,E1 24411.216,E2 24411.216} C_VEL
LIN {X 0,Y 665.317,Z 1146.012,A -85,B 0,C 180,E1 24409.398,E2 24409.398} C_VEL
LIN {X 0,Y 664.82,Z 1158.887,A -85,B 0,C 180,E1 24407.235,E2 24407.235} C_VEL
LIN {X 0,Y 664.423,Z 1170.661,A -85,B 0,C 180,E1 24404.912,E2 24404.912} C_VEL
LIN {X 0,Y 664.223,Z 1178.795,A -85,B 0,C 180,E1 24403.05,E2 24403.05} C_VEL
LIN {X 0,Y 664.054,Z 1186.417,A -85,B 0,C 180,E1 24401.025,E2 24401.025} C_VEL
LIN {X 0,Y 663.977,Z 1193.594,A -85,B 0,C 180,E1 24398.661,E2 24398.661} C_VEL
LIN {X 0,Y 663.931,Z 1198.969,A -85,B 0,C 180,E1 24396.292,E2 24396.292} C_VEL
LIN {X 0,Y 663.915,Z 1202.481,A -85,B 0,C 180,E1 24394.059,E2 24394.059} C_VEL
LIN {X 0,Y 663.907,Z 1204.549,A -85,B 0,C 180,E1 24391.726,E2 24391.726} C_VEL
LIN {X 0,Y 663.891,Z 1204.872,A -85,B 0,C 180,E1 24389.483,E2 24389.483} C_VEL
LIN {X 0,Y 663.908,Z 1203.95,A -85,B 0,C 180,E1 24387.411,E2 24387.411} C_VEL
LIN {X 0,Y 663.917,Z 1201.428,A -85,B 0,C 180,E1 24385.162,E2 24385.162} C_VEL
LIN {X 0,Y 663.948,Z 1197.152,A -85,B 0,C 180,E1 24382.82,E2 24382.82} C_VEL
LIN {X 0,Y 664.001,Z 1191.281,A -85,B 0,C 180,E1 24380.519,E2 24380.519} C_VEL
LIN {X 0,Y 664.11,Z 1183.96,A -85,B 0,C 180,E1 24378.273,E2 24378.273} C_VEL
LIN {X 0,Y 664.345,Z 1173.757,A -85,B 0,C 180,E1 24375.76,E2 24375.76} C_VEL
LIN {X 0,Y 664.618,Z 1164.076,A -85,B 0,C 180,E1 24373.751,E2 24373.751} C_VEL
LIN {X 0,Y 665.01,Z 1153.634,A -85,B 0,C 180,E1 24371.853,E2 24371.853} C_VEL
LIN {X 0,Y 665.631,Z 1139.567,A -85,B 0,C 180,E1 24369.605,E2 24369.605} C_VEL
LIN {X 0,Y 666.364,Z 1124.403,A -85,B 0,C 180,E1 24367.504,E2 24367.504} C_VEL
LIN {X 0,Y 667.166,Z 1109.515,A -85,B 0,C 180,E1 24365.661,E2 24365.661} C_VEL
LIN {X 0,Y 668.347,Z 1090.658,A -85,B 0,C 180,E1 24363.583,E2 24363.583} C_VEL
LIN {X 0,Y 669.435,Z 1073.311,A -85,B 0,C 180,E1 24361.886,E2 24361.886} C_VEL
LIN {X 0,Y 670.618,Z 1056.205,A -85,B 0,C 180,E1 24360.372,E2 24360.372} C_VEL
LIN {X 0,Y 672.189,Z 1034.205,A -85,B 0,C 180,E1 24358.627,E2 24358.627} C_VEL
LIN {X 0,Y 673.617,Z 1013.162,A -85,B 0,C 180,E1 24357.156,E2 24357.156} C_VEL
LIN {X 0,Y 674.997,Z 993.058,A -85,B 0,C 180,E1 24355.901,E2 24355.901} C_VEL
LIN {X 0,Y 676.708,Z 968.655,A -85,B 0,C 180,E1 24354.554,E2 24354.554} C_VEL
LIN {X 0,Y 678.238,Z 943.99,A -85,B 0,C 180,E1 24353.393,E2 24353.393} C_VEL
LIN {X 0,Y 679.403,Z 923.887,A -85,B 0,C 180,E1 24352.569,E2 24352.569} C_VEL
LIN {X 0,Y 680.471,Z 903.03,A -85,B 0,C 180,E1 24351.826,E2 24351.826} C_VEL
LIN {X 0,Y 681.604,Z 879.622,A -85,B 0,C 180,E1 24351.122,E2 24351.122} C_VEL
LIN {X 0,Y 682.719,Z 851.782,A -85,B 0,C 180,E1 24350.464,E2 24350.464} C_VEL
LIN {X 0,Y 683.44,Z 826.248,A -85,B 0,C 180,E1 24350.021,E2 24350.021} C_VEL
LIN {X 0,Y 686.306,Z 607.969,A -85,B 0,C 180,E1 24347.22,E2 24347.22} C_VEL
LIN {X 0,Y 689.077,Z 403.56,A -85,B 0,C 180,E1 24344.531,E2 24344.531} C_VEL
LIN {X 0,Y 689.288,Z 376.406,A -85,B 0,C 180,E1 24344.152,E2 24344.152} C_VEL
LIN {X 0,Y 687.98,Z 372.02,A -85,B 0,C 180,E1 24343.976,E2 24343.976} C_VEL
LIN {X 0,Y 677.361,Z 356.315,A -85,B 0,C 180,E1 24342.797,E2 24342.797} C_VEL
LIN {X 0,Y 673.311,Z 350.327,A -85,B 0,C 180,E1 24342.309,E2 24342.309} C_VEL
LIN {X 0,Y 666.325,Z 335.437,A -85,B 0,C 180,E1 24340.411,E2 24340.411} C_VEL
LIN {X 0,Y 664.698,Z 332.123,A -85,B 0,C 180,E1 24339.966,E2 24339.966} C_VEL
LIN {X 0,Y 664.576,Z 331.449,A -85,B 0,C 180,E1 24339.862,E2 24339.862} C_VEL
LIN {X 0,Y 664.564,Z 331.447,A -85,B 0,C 180,E1 24337.259,E2 24337.259} C_VEL
LIN {X 0,Y 664.638,Z 331.443,A -85,B 0,C 180,E1 24334.32,E2 24334.32} C_VEL
LIN {X 0,Y 664.556,Z 331.438,A -85,B 0,C 180,E1 24331.451,E2 24331.451} C_VEL
LIN {X 0,Y 664.557,Z 331.445,A -85,B 0,C 180,E1 24328.979,E2 24328.979} C_VEL
LIN {X 0,Y 664.626,Z 331.422,A -85,B 0,C 180,E1 24326.059,E2 24326.059} C_VEL
LIN {X 0,Y 664.547,Z 331.445,A -85,B 0,C 180,E1 24323.217,E2 24323.217} C_VEL
LIN {X 0,Y 664.548,Z 331.433,A -85,B 0,C 180,E1 24320.799,E2 24320.799} C_VEL
LIN {X 0,Y 664.605,Z 331.43,A -85,B 0,C 180,E1 24317.783,E2 24317.783} C_VEL
LIN {X 0,Y 664.538,Z 331.445,A -85,B 0,C 180,E1 24314.993,E2 24314.993} C_VEL
LIN {X 0,Y 664.556,Z 331.443,A -85,B 0,C 180,E1 24312.456,E2 24312.456} C_VEL
LIN {X 0,Y 664.564,Z 331.448,A -85,B 0,C 180,E1 24309.255,E2 24309.255} C_VEL
LIN {X 0,Y 664.544,Z 331.436,A -85,B 0,C 180,E1 24306.74,E2 24306.74} C_VEL
LIN {X 0,Y 664.585,Z 331.438,A -85,B 0,C 180,E1 24304.055,E2 24304.055} C_VEL
LIN {X 0,Y 664.563,Z 331.426,A -85,B 0,C 180,E1 24300.948,E2 24300.948} C_VEL
LIN {X 0,Y 664.554,Z 331.442,A -85,B 0,C 180,E1 24298.448,E2 24298.448} C_VEL
LIN {X 0,Y 664.63,Z 331.423,A -85,B 0,C 180,E1 24295.6,E2 24295.6} C_VEL
LIN {X 0,Y 664.567,Z 331.445,A -85,B 0,C 180,E1 24292.652,E2 24292.652} C_VEL
LIN {X 0,Y 664.565,Z 331.434,A -85,B 0,C 180,E1 24290.124,E2 24290.124} C_VEL
LIN {X 0,Y 664.64,Z 331.442,A -85,B 0,C 180,E1 24287.119,E2 24287.119} C_VEL
LIN {X 0,Y 664.565,Z 331.419,A -85,B 0,C 180,E1 24284.287,E2 24284.287} C_VEL
LIN {X 0,Y 664.603,Z 331.446,A -85,B 0,C 180,E1 24281.582,E2 24281.582} C_VEL
LIN {X 0,Y 664.589,Z 331.441,A -85,B 0,C 180,E1 24278.463,E2 24278.463} C_VEL
LIN {X 0,Y 664.577,Z 331.434,A -85,B 0,C 180,E1 24275.843,E2 24275.843} C_VEL
LIN {X 0,Y 664.651,Z 331.438,A -85,B 0,C 180,E1 24272.882,E2 24272.882} C_VEL
LIN {X 0,Y 664.58,Z 331.441,A -85,B 0,C 180,E1 24269.933,E2 24269.933} C_VEL
LIN {X 0,Y 664.634,Z 331.444,A -85,B 0,C 180,E1 24267.082,E2 24267.082} C_VEL
LIN {X 0,Y 664.632,Z 331.607,A -85,B 0,C 180,E1 24265.262,E2 24265.262} C_VEL
LIN {X 0,Y 666.123,Z 335.167,A -85,B 0,C 180,E1 24264.802,E2 24264.802} C_VEL
LIN {X 0,Y 666.809,Z 336.494,A -85,B 0,C 180,E1 24264.619,E2 24264.619} C_VEL
LIN {X 0,Y 668.098,Z 341.072,A -85,B 0,C 180,E1 24264.219,E2 24264.219} C_VEL
LIN {X 0,Y 670.66,Z 350.294,A -85,B 0,C 180,E1 24263.719,E2 24263.719} C_VEL
LIN {X 0,Y 674.032,Z 359.61,A -85,B 0,C 180,E1 24263.26,E2 24263.26} C_VEL
LIN {X 0,Y 676.816,Z 364.333,A -85,B 0,C 180,E1 24262.933,E2 24262.933} C_VEL
LIN {X 0,Y 683.778,Z 375.129,A -85,B 0,C 180,E1 24262.15,E2 24262.15} C_VEL
LIN {X 0,Y 680.457,Z 596.265,A -85,B 0,C 180,E1 24259.216,E2 24259.216} C_VEL
LIN {X 0,Y 677.335,Z 814.821,A -85,B 0,C 180,E1 24256.391,E2 24256.391} C_VEL
LIN {X 0,Y 676.601,Z 838.587,A -85,B 0,C 180,E1 24255.988,E2 24255.988} C_VEL
LIN {X 0,Y 675.551,Z 865.236,A -85,B 0,C 180,E1 24255.383,E2 24255.383} C_VEL
LIN {X 0,Y 674.23,Z 890.653,A -85,B 0,C 180,E1 24254.634,E2 24254.634} C_VEL
LIN {X 0,Y 673.07,Z 911.387,A -85,B 0,C 180,E1 24253.904,E2 24253.904} C_VEL
LIN {X 0,Y 671.845,Z 930.794,A -85,B 0,C 180,E1 24253.119,E2 24253.119} C_VEL
LIN {X 0,Y 670.495,Z 950.734,A -85,B 0,C 180,E1 24252.2,E2 24252.2} C_VEL
LIN {X 0,Y 669.022,Z 971.514,A -85,B 0,C 180,E1 24251.116,E2 24251.116} C_VEL
LIN {X 0,Y 667.146,Z 996.683,A -85,B 0,C 180,E1 24249.613,E2 24249.613} C_VEL
LIN {X 0,Y 665.518,Z 1017.289,A -85,B 0,C 180,E1 24248.208,E2 24248.208} C_VEL
LIN {X 0,Y 664.116,Z 1035.636,A -85,B 0,C 180,E1 24246.813,E2 24246.813} C_VEL
LIN {X 0,Y 662.605,Z 1056.563,A -85,B 0,C 180,E1 24245.042,E2 24245.042} C_VEL
LIN {X 0,Y 661.154,Z 1075.805,A -85,B 0,C 180,E1 24243.192,E2 24243.192} C_VEL
LIN {X 0,Y 660.048,Z 1091.905,A -85,B 0,C 180,E1 24241.474,E2 24241.474} C_VEL
LIN {X 0,Y 658.869,Z 1110.54,A -85,B 0,C 180,E1 24239.236,E2 24239.236} C_VEL
LIN {X 0,Y 658.056,Z 1124.664,A -85,B 0,C 180,E1 24237.314,E2 24237.314} C_VEL
LIN {X 0,Y 657.405,Z 1137.849,A -85,B 0,C 180,E1 24235.301,E2 24235.301} C_VEL
LIN {X 0,Y 656.801,Z 1151.429,A -85,B 0,C 180,E1 24232.922,E2 24232.922} C_VEL
LIN {X 0,Y 656.472,Z 1161.451,A -85,B 0,C 180,E1 24230.879,E2 24230.879} C_VEL
LIN {X 0,Y 656.238,Z 1169.714,A -85,B 0,C 180,E1 24228.937,E2 24228.937} C_VEL
LIN {X 0,Y 656.066,Z 1177.659,A -85,B 0,C 180,E1 24226.741,E2 24226.741} C_VEL
LIN {X 0,Y 655.975,Z 1184.434,A -85,B 0,C 180,E1 24224.386,E2 24224.386} C_VEL
LIN {X 0,Y 655.927,Z 1189.296,A -85,B 0,C 180,E1 24222.143,E2 24222.143} C_VEL
LIN {X 0,Y 655.91,Z 1192.651,A -85,B 0,C 180,E1 24219.919,E2 24219.919} C_VEL
LIN {X 0,Y 655.907,Z 1194.577,A -85,B 0,C 180,E1 24217.621,E2 24217.621} C_VEL
LIN {X 0,Y 655.896,Z 1194.87,A -85,B 0,C 180,E1 24215.423,E2 24215.423} C_VEL
LIN {X 0,Y 655.908,Z 1193.937,A -85,B 0,C 180,E1 24213.321,E2 24213.321} C_VEL
LIN {X 0,Y 655.919,Z 1191.414,A -85,B 0,C 180,E1 24211.048,E2 24211.048} C_VEL
LIN {X 0,Y 655.949,Z 1187.157,A -85,B 0,C 180,E1 24208.689,E2 24208.689} C_VEL
LIN {X 0,Y 656.006,Z 1181.447,A -85,B 0,C 180,E1 24206.417,E2 24206.417} C_VEL
LIN {X 0,Y 656.136,Z 1174.163,A -85,B 0,C 180,E1 24204.14,E2 24204.14} C_VEL
LIN {X 0,Y 656.389,Z 1163.99,A -85,B 0,C 180,E1 24201.591,E2 24201.591} C_VEL
LIN {X 0,Y 656.701,Z 1154.368,A -85,B 0,C 180,E1 24199.561,E2 24199.561} C_VEL
LIN {X 0,Y 657.106,Z 1143.796,A -85,B 0,C 180,E1 24197.611,E2 24197.611} C_VEL
LIN {X 0,Y 657.785,Z 1130.093,A -85,B 0,C 180,E1 24195.384,E2 24195.384} C_VEL
LIN {X 0,Y 658.612,Z 1114.819,A -85,B 0,C 180,E1 24193.235,E2 24193.235} C_VEL
LIN {X 0,Y 659.509,Z 1099.936,A -85,B 0,C 180,E1 24191.365,E2 24191.365} C_VEL
LIN {X 0,Y 660.79,Z 1081.033,A -85,B 0,C 180,E1 24189.252,E2 24189.252} C_VEL
LIN {X 0,Y 662.057,Z 1063.095,A -85,B 0,C 180,E1 24187.477,E2 24187.477} C_VEL
LIN {X 0,Y 663.414,Z 1045.31,A -85,B 0,C 180,E1 24185.893,E2 24185.893} C_VEL
LIN {X 0,Y 665.172,Z 1022.205,A -85,B 0,C 180,E1 24184.06,E2 24184.06} C_VEL
LIN {X 0,Y 666.647,Z 1002.534,A -85,B 0,C 180,E1 24182.68,E2 24182.68} C_VEL
LIN {X 0,Y 668.156,Z 982.734,A -85,B 0,C 180,E1 24181.437,E2 24181.437} C_VEL
LIN {X 0,Y 669.995,Z 958.7,A -85,B 0,C 180,E1 24180.102,E2 24180.102} C_VEL
LIN {X 0,Y 671.629,Z 934.319,A -85,B 0,C 180,E1 24178.946,E2 24178.946} C_VEL
LIN {X 0,Y 672.831,Z 915.378,A -85,B 0,C 180,E1 24178.159,E2 24178.159} C_VEL
LIN {X 0,Y 673.974,Z 894.91,A -85,B 0,C 180,E1 24177.416,E2 24177.416} C_VEL
LIN {X 0,Y 675.17,Z 872.592,A -85,B 0,C 180,E1 24176.729,E2 24176.729} C_VEL
LIN {X 0,Y 676.386,Z 845.641,A -85,B 0,C 180,E1 24176.063,E2 24176.063} C_VEL
LIN {X 0,Y 677.23,Z 819.011,A -85,B 0,C 180,E1 24175.581,E2 24175.581} C_VEL
LIN {X 0,Y 678.754,Z 717.655,A -85,B 0,C 180,E1 24174.266,E2 24174.266} C_VEL
LIN {X 0,Y 681.692,Z 509.547,A -85,B 0,C 180,E1 24171.552,E2 24171.552} C_VEL
LIN {X 0,Y 683.713,Z 374.653,A -85,B 0,C 180,E1 24169.747,E2 24169.747} C_VEL
LIN {X 0,Y 668.596,Z 352.366,A -85,B 0,C 180,E1 24168.028,E2 24168.028} C_VEL
LIN {X 0,Y 660.77,Z 341.195,A -85,B 0,C 180,E1 24167.088,E2 24167.088} C_VEL
LIN {X 0,Y 657.933,Z 335.842,A -85,B 0,C 180,E1 24166.336,E2 24166.336} C_VEL
LIN {X 0,Y 656.703,Z 332.433,A -85,B 0,C 180,E1 24165.873,E2 24165.873} C_VEL
LIN {X 0,Y 656.69,Z 332.433,A -85,B 0,C 180,E1 24162.654,E2 24162.654} C_VEL
LIN {X 0,Y 656.707,Z 332.429,A -85,B 0,C 180,E1 24159.609,E2 24159.609} C_VEL
LIN {X 0,Y 656.681,Z 332.433,A -85,B 0,C 180,E1 24156.491,E2 24156.491} C_VEL
LIN {X 0,Y 656.703,Z 332.427,A -85,B 0,C 180,E1 24153.448,E2 24153.448} C_VEL
LIN {X 0,Y 656.672,Z 332.43,A -85,B 0,C 180,E1 24150.306,E2 24150.306} C_VEL
LIN {X 0,Y 656.694,Z 332.412,A -85,B 0,C 180,E1 24147.376,E2 24147.376} C_VEL
LIN {X 0,Y 656.668,Z 332.434,A -85,B 0,C 180,E1 24144.207,E2 24144.207} C_VEL
LIN {X 0,Y 656.677,Z 332.414,A -85,B 0,C 180,E1 24141.341,E2 24141.341} C_VEL
LIN {X 0,Y 656.67,Z 332.431,A -85,B 0,C 180,E1 24138.17,E2 24138.17} C_VEL
LIN {X 0,Y 656.659,Z 332.421,A -85,B 0,C 180,E1 24135.364,E2 24135.364} C_VEL
LIN {X 0,Y 656.673,Z 332.416,A -85,B 0,C 180,E1 24132.167,E2 24132.167} C_VEL
LIN {X 0,Y 656.646,Z 332.428,A -85,B 0,C 180,E1 24129.35,E2 24129.35} C_VEL
LIN {X 0,Y 656.7,Z 332.429,A -85,B 0,C 180,E1 24126.294,E2 24126.294} C_VEL
LIN {X 0,Y 656.634,Z 332.433,A -85,B 0,C 180,E1 24123.405,E2 24123.405} C_VEL
LIN {X 0,Y 656.712,Z 332.425,A -85,B 0,C 180,E1 24120.436,E2 24120.436} C_VEL
LIN {X 0,Y 656.629,Z 332.432,A -85,B 0,C 180,E1 24117.469,E2 24117.469} C_VEL
LIN {X 0,Y 656.648,Z 332.428,A -85,B 0,C 180,E1 24114.758,E2 24114.758} C_VEL
LIN {X 0,Y 656.636,Z 332.428,A -85,B 0,C 180,E1 24111.594,E2 24111.594} C_VEL
LIN {X 0,Y 656.617,Z 332.434,A -85,B 0,C 180,E1 24109.027,E2 24109.027} C_VEL
LIN {X 0,Y 656.701,Z 332.399,A -85,B 0,C 180,E1 24106.08,E2 24106.08} C_VEL
LIN {X 0,Y 656.612,Z 332.436,A -85,B 0,C 180,E1 24103.182,E2 24103.182} C_VEL
LIN {X 0,Y 656.614,Z 332.411,A -85,B 0,C 180,E1 24100.612,E2 24100.612} C_VEL
LIN {X 0,Y 656.646,Z 332.436,A -85,B 0,C 180,E1 24097.53,E2 24097.53} C_VEL
LIN {X 0,Y 656.599,Z 332.407,A -85,B 0,C 180,E1 24094.857,E2 24094.857} C_VEL
LIN {X 0,Y 656.645,Z 332.437,A -85,B 0,C 180,E1 24092.129,E2 24092.129} C_VEL
LIN {X 0,Y 656.621,Z 332.431,A -85,B 0,C 180,E1 24089.022,E2 24089.022} C_VEL
LIN {X 0,Y 656.62,Z 332.439,A -85,B 0,C 180,E1 24086.403,E2 24086.403} C_VEL
LIN {X 0,Y 656.681,Z 332.434,A -85,B 0,C 180,E1 24083.353,E2 24083.353} C_VEL
LIN {X 0,Y 656.643,Z 332.517,A -85,B 0,C 180,E1 24080.837,E2 24080.837} C_VEL
LIN {X 0,Y 657.96,Z 335.975,A -85,B 0,C 180,E1 24080.396,E2 24080.396} C_VEL
LIN {X 0,Y 659.116,Z 338.231,A -85,B 0,C 180,E1 24080.081,E2 24080.081} C_VEL
LIN {X 0,Y 661.379,Z 342.904,A -85,B 0,C 180,E1 24079.452,E2 24079.452} C_VEL
LIN {X 0,Y 665.397,Z 351.085,A -85,B 0,C 180,E1 24078.408,E2 24078.408} C_VEL
LIN {X 0,Y 680.915,Z 373.533,A -85,B 0,C 180,E1 24076.621,E2 24076.621} C_VEL
LIN {X 0,Y 683.516,Z 378.01,A -85,B 0,C 180,E1 24076.324,E2 24076.324} C_VEL
LIN {X 0,Y 683.818,Z 380.657,A -85,B 0,C 180,E1 24076.258,E2 24076.258} C_VEL
LIN {X 0,Y 680.667,Z 591.328,A -85,B 0,C 180,E1 24073.457,E2 24073.457} C_VEL
LIN {X 0,Y 677.585,Z 814.354,A -85,B 0,C 180,E1 24070.581,E2 24070.581} C_VEL
LIN {X 0,Y 676.829,Z 842.187,A -85,B 0,C 180,E1 24070.154,E2 24070.154} C_VEL
LIN {X 0,Y 675.924,Z 865.91,A -85,B 0,C 180,E1 24069.656,E2 24069.656} C_VEL
LIN {X 0,Y 674.732,Z 891.752,A -85,B 0,C 180,E1 24068.964,E2 24068.964} C_VEL
LIN {X 0,Y 673.229,Z 918.726,A -85,B 0,C 180,E1 24068.051,E2 24068.051} C_VEL
LIN {X 0,Y 671.901,Z 939.829,A -85,B 0,C 180,E1 24067.206,E2 24067.206} C_VEL
LIN {X 0,Y 670.503,Z 960.706,A -85,B 0,C 180,E1 24066.248,E2 24066.248} C_VEL
LIN {X 0,Y 668.873,Z 983.888,A -85,B 0,C 180,E1 24065.032,E2 24065.032} C_VEL
LIN {X 0,Y 666.981,Z 1008.53,A -85,B 0,C 180,E1 24063.538,E2 24063.538} C_VEL
LIN {X 0,Y 665.452,Z 1028.172,A -85,B 0,C 180,E1 24062.19,E2 24062.19} C_VEL
LIN {X 0,Y 663.951,Z 1048.284,A -85,B 0,C 180,E1 24060.648,E2 24060.648} C_VEL
LIN {X 0,Y 662.313,Z 1070.047,A -85,B 0,C 180,E1 24058.76,E2 24058.76} C_VEL
LIN {X 0,Y 661.058,Z 1086.845,A -85,B 0,C 180,E1 24057.132,E2 24057.132} C_VEL
LIN {X 0,Y 659.906,Z 1104.465,A -85,B 0,C 180,E1 24055.233,E2 24055.233} C_VEL
LIN {X 0,Y 658.774,Z 1121.891,A -85,B 0,C 180,E1 24053.104,E2 24053.104} C_VEL
LIN {X 0,Y 658.001,Z 1135.749,A -85,B 0,C 180,E1 24051.202,E2 24051.202} C_VEL
LIN {X 0,Y 657.305,Z 1150.027,A -85,B 0,C 180,E1 24048.998,E2 24048.998} C_VEL
LIN {X 0,Y 656.753,Z 1162.675,A -85,B 0,C 180,E1 24046.723,E2 24046.723} C_VEL
LIN {X 0,Y 656.451,Z 1171.894,A -85,B 0,C 180,E1 24044.827,E2 24044.827} C_VEL
LIN {X 0,Y 656.232,Z 1179.869,A -85,B 0,C 180,E1 24042.943,E2 24042.943} C_VEL
LIN {X 0,Y 656.05,Z 1187.891,A -85,B 0,C 180,E1 24040.716,E2 24040.716} C_VEL
LIN {X 0,Y 655.969,Z 1194.693,A -85,B 0,C 180,E1 24038.326,E2 24038.326} C_VEL
LIN {X 0,Y 655.929,Z 1199.409,A -85,B 0,C 180,E1 24036.126,E2 24036.126} C_VEL
LIN {X 0,Y 655.91,Z 1202.789,A -85,B 0,C 180,E1 24033.846,E2 24033.846} C_VEL
LIN {X 0,Y 655.911,Z 1204.624,A -85,B 0,C 180,E1 24031.485,E2 24031.485} C_VEL
LIN {X 0,Y 655.893,Z 1204.849,A -85,B 0,C 180,E1 24029.389,E2 24029.389} C_VEL
LIN {X 0,Y 655.909,Z 1203.947,A -85,B 0,C 180,E1 24027.379,E2 24027.379} C_VEL
LIN {X 0,Y 655.92,Z 1201.428,A -85,B 0,C 180,E1 24025.103,E2 24025.103} C_VEL
LIN {X 0,Y 655.949,Z 1197.152,A -85,B 0,C 180,E1 24022.732,E2 24022.732} C_VEL
LIN {X 0,Y 656.009,Z 1191.376,A -85,B 0,C 180,E1 24020.437,E2 24020.437} C_VEL
LIN {X 0,Y 656.126,Z 1184.279,A -85,B 0,C 180,E1 24018.217,E2 24018.217} C_VEL
LIN {X 0,Y 656.39,Z 1174.089,A -85,B 0,C 180,E1 24015.658,E2 24015.658} C_VEL
LIN {X 0,Y 656.694,Z 1164.274,A -85,B 0,C 180,E1 24013.587,E2 24013.587} C_VEL
LIN {X 0,Y 657.113,Z 1154.136,A -85,B 0,C 180,E1 24011.715,E2 24011.715} C_VEL
LIN {X 0,Y 657.764,Z 1140.78,A -85,B 0,C 180,E1 24009.536,E2 24009.536} C_VEL
LIN {X 0,Y 658.599,Z 1125.104,A -85,B 0,C 180,E1 24007.318,E2 24007.318} C_VEL
LIN {X 0,Y 659.476,Z 1110.398,A -85,B 0,C 180,E1 24005.466,E2 24005.466} C_VEL
LIN {X 0,Y 660.729,Z 1092.314,A -85,B 0,C 180,E1 24003.428,E2 24003.428} C_VEL
LIN {X 0,Y 662.001,Z 1073.817,A -85,B 0,C 180,E1 24001.591,E2 24001.591} C_VEL
LIN {X 0,Y 663.29,Z 1056.84,A -85,B 0,C 180,E1 24000.069,E2 24000.069} C_VEL
LIN {X 0,Y 664.963,Z 1035.527,A -85,B 0,C 180,E1 23998.347,E2 23998.347} C_VEL
LIN {X 0,Y 666.619,Z 1013,A -85,B 0,C 180,E1 23996.755,E2 23996.755} C_VEL
LIN {X 0,Y 668.13,Z 993.018,A -85,B 0,C 180,E1 23995.498,E2 23995.498} C_VEL
LIN {X 0,Y 669.973,Z 968.962,A -85,B 0,C 180,E1 23994.161,E2 23994.161} C_VEL
LIN {X 0,Y 671.663,Z 943.882,A -85,B 0,C 180,E1 23992.97,E2 23992.97} C_VEL
LIN {X 0,Y 672.974,Z 923.051,A -85,B 0,C 180,E1 23992.114,E2 23992.114} C_VEL
LIN {X 0,Y 674.098,Z 902.832,A -85,B 0,C 180,E1 23991.392,E2 23991.392} C_VEL
LIN {X 0,Y 675.312,Z 879.644,A -85,B 0,C 180,E1 23990.692,E2 23990.692} C_VEL
LIN {X 0,Y 676.521,Z 851.783,A -85,B 0,C 180,E1 23990.029,E2 23990.029} C_VEL
LIN {X 0,Y 677.297,Z 826.323,A -85,B 0,C 180,E1 23989.586,E2 23989.586} C_VEL
LIN {X 0,Y 680.392,Z 610.618,A -85,B 0,C 180,E1 23986.796,E2 23986.796} C_VEL
LIN {X 0,Y 683.423,Z 406.015,A -85,B 0,C 180,E1 23984.083,E2 23984.083} C_VEL
LIN {X 0,Y 683.694,Z 378.681,A -85,B 0,C 180,E1 23983.701,E2 23983.701} C_VEL
LIN {X 0,Y 682.678,Z 376.231,A -85,B 0,C 180,E1 23983.575,E2 23983.575} C_VEL
LIN {X 0,Y 669.174,Z 356.396,A -85,B 0,C 180,E1 23982.038,E2 23982.038} C_VEL
LIN {X 0,Y 664.935,Z 350.183,A -85,B 0,C 180,E1 23981.51,E2 23981.51} C_VEL
LIN {X 0,Y 660.086,Z 340.176,A -85,B 0,C 180,E1 23980.188,E2 23980.188} C_VEL
LIN {X 0,Y 658.149,Z 336.23,A -85,B 0,C 180,E1 23979.649,E2 23979.649} C_VEL
LIN {X 0,Y 656.678,Z 332.745,A -85,B 0,C 180,E1 23979.191,E2 23979.191} C_VEL
LIN {X 0,Y 656.642,Z 332.44,A -85,B 0,C 180,E1 23979.052,E2 23979.052} C_VEL
LIN {X 0,Y 656.644,Z 332.431,A -85,B 0,C 180,E1 23975.892,E2 23975.892} C_VEL
LIN {X 0,Y 656.62,Z 332.435,A -85,B 0,C 180,E1 23973.244,E2 23973.244} C_VEL
LIN {X 0,Y 656.709,Z 332.407,A -85,B 0,C 180,E1 23970.263,E2 23970.263} C_VEL
LIN {X 0,Y 656.615,Z 332.427,A -85,B 0,C 180,E1 23967.38,E2 23967.38} C_VEL
LIN {X 0,Y 656.624,Z 332.431,A -85,B 0,C 180,E1 23964.757,E2 23964.757} C_VEL
LIN {X 0,Y 656.625,Z 332.414,A -85,B 0,C 180,E1 23961.53,E2 23961.53} C_VEL
LIN {X 0,Y 656.604,Z 332.438,A -85,B 0,C 180,E1 23958.927,E2 23958.927} C_VEL
LIN {X 0,Y 656.686,Z 332.408,A -85,B 0,C 180,E1 23955.998,E2 23955.998} C_VEL
LIN {X 0,Y 656.606,Z 332.433,A -85,B 0,C 180,E1 23953.115,E2 23953.115} C_VEL
LIN {X 0,Y 656.61,Z 332.417,A -85,B 0,C 180,E1 23950.529,E2 23950.529} C_VEL
LIN {X 0,Y 656.656,Z 332.424,A -85,B 0,C 180,E1 23947.437,E2 23947.437} C_VEL
LIN {X 0,Y 656.608,Z 332.426,A -85,B 0,C 180,E1 23944.717,E2 23944.717} C_VEL
LIN {X 0,Y 656.649,Z 332.433,A -85,B 0,C 180,E1 23942.007,E2 23942.007} C_VEL
LIN {X 0,Y 656.632,Z 332.43,A -85,B 0,C 180,E1 23938.953,E2 23938.953} C_VEL
LIN {X 0,Y 656.618,Z 332.433,A -85,B 0,C 180,E1 23936.333,E2 23936.333} C_VEL
LIN {X 0,Y 656.707,Z 332.417,A -85,B 0,C 180,E1 23933.355,E2 23933.355} C_VEL
LIN {X 0,Y 656.623,Z 332.424,A -85,B 0,C 180,E1 23930.446,E2 23930.446} C_VEL
LIN {X 0,Y 656.661,Z 332.426,A -85,B 0,C 180,E1 23927.691,E2 23927.691} C_VEL
LIN {X 0,Y 656.639,Z 332.406,A -85,B 0,C 180,E1 23924.545,E2 23924.545} C_VEL
LIN {X 0,Y 656.637,Z 332.434,A -85,B 0,C 180,E1 23921.902,E2 23921.902} C_VEL
LIN {X 0,Y 656.694,Z 332.414,A -85,B 0,C 180,E1 23918.847,E2 23918.847} C_VEL
LIN {X 0,Y 656.635,Z 332.424,A -85,B 0,C 180,E1 23916.01,E2 23916.01} C_VEL
LIN {X 0,Y 656.705,Z 332.432,A -85,B 0,C 180,E1 23913.114,E2 23913.114} C_VEL
LIN {X 0,Y 656.648,Z 332.429,A -85,B 0,C 180,E1 23910.137,E2 23910.137} C_VEL
LIN {X 0,Y 656.663,Z 332.436,A -85,B 0,C 180,E1 23907.382,E2 23907.382} C_VEL
LIN {X 0,Y 656.665,Z 332.532,A -85,B 0,C 180,E1 23906.006,E2 23906.006} C_VEL
LIN {X 0,Y 657.933,Z 335.884,A -85,B 0,C 180,E1 23905.573,E2 23905.573} C_VEL
LIN {X 0,Y 658.923,Z 337.634,A -85,B 0,C 180,E1 23905.316,E2 23905.316} C_VEL
LIN {X 0,Y 660.994,Z 341.62,A -85,B 0,C 180,E1 23904.793,E2 23904.793} C_VEL
LIN {X 0,Y 674.936,Z 361.727,A -85,B 0,C 180,E1 23903.144,E2 23903.144} C_VEL
LIN {X 0,Y 676.816,Z 364.333,A -85,B 0,C 180,E1 23902.933,E2 23902.933} C_VEL
LIN {X 0,Y 678.471,Z 367.552,A -85,B 0,C 180,E1 23902.734,E2 23902.734} C_VEL
LIN {X 0,Y 679.505,Z 372.542,A -85,B 0,C 180,E1 23902.566,E2 23902.566} C_VEL
LIN {X 0,Y 679.572,Z 380.245,A -85,B 0,C 180,E1 23902.444,E2 23902.444} C_VEL
LIN {X 0,Y 677.859,Z 398.319,A -85,B 0,C 180,E1 23902.325,E2 23902.325} C_VEL
LIN {X 0,Y 677.826,Z 399.518,A -85,B 0,C 180,E1 23902.309,E2 23902.309} C_VEL
LIN {X 0,Y 674.088,Z 630.816,A -85,B 0,C 180,E1 23899.23,E2 23899.23} C_VEL
LIN {X 0,Y 671.156,Z 818.019,A -85,B 0,C 180,E1 23896.788,E2 23896.788} C_VEL
LIN {X 0,Y 670.293,Z 843.616,A -85,B 0,C 180,E1 23896.33,E2 23896.33} C_VEL
LIN {X 0,Y 668.979,Z 871.149,A -85,B 0,C 180,E1 23895.661,E2 23895.661} C_VEL
LIN {X 0,Y 667.713,Z 893.541,A -85,B 0,C 180,E1 23894.975,E2 23894.975} C_VEL
LIN {X 0,Y 666.52,Z 913.242,A -85,B 0,C 180,E1 23894.264,E2 23894.264} C_VEL
LIN {X 0,Y 665.159,Z 933.151,A -85,B 0,C 180,E1 23893.442,E2 23893.442} C_VEL
LIN {X 0,Y 663.562,Z 955.039,A -85,B 0,C 180,E1 23892.408,E2 23892.408} C_VEL
LIN {X 0,Y 661.51,Z 980.827,A -85,B 0,C 180,E1 23890.994,E2 23890.994} C_VEL
LIN {X 0,Y 659.788,Z 1001.446,A -85,B 0,C 180,E1 23889.699,E2 23889.699} C_VEL
LIN {X 0,Y 658.187,Z 1020.558,A -85,B 0,C 180,E1 23888.357,E2 23888.357} C_VEL
LIN {X 0,Y 656.393,Z 1042.801,A -85,B 0,C 180,E1 23886.603,E2 23886.603} C_VEL
LIN {X 0,Y 654.829,Z 1061.661,A -85,B 0,C 180,E1 23884.918,E2 23884.918} C_VEL
LIN {X 0,Y 653.488,Z 1078.364,A -85,B 0,C 180,E1 23883.265,E2 23883.265} C_VEL
LIN {X 0,Y 652.122,Z 1097.249,A -85,B 0,C 180,E1 23881.176,E2 23881.176} C_VEL
LIN {X 0,Y 650.984,Z 1113.496,A -85,B 0,C 180,E1 23879.136,E2 23879.136} C_VEL
LIN {X 0,Y 650.128,Z 1127.413,A -85,B 0,C 180,E1 23877.179,E2 23877.179} C_VEL
LIN {X 0,Y 649.357,Z 1141.946,A -85,B 0,C 180,E1 23874.857,E2 23874.857} C_VEL
LIN {X 0,Y 648.813,Z 1153.354,A -85,B 0,C 180,E1 23872.756,E2 23872.756} C_VEL
LIN {X 0,Y 648.504,Z 1162.363,A -85,B 0,C 180,E1 23870.864,E2 23870.864} C_VEL
LIN {X 0,Y 648.246,Z 1170.861,A -85,B 0,C 180,E1 23868.806,E2 23868.806} C_VEL
LIN {X 0,Y 648.068,Z 1178.881,A -85,B 0,C 180,E1 23866.492,E2 23866.492} C_VEL
LIN {X 0,Y 647.968,Z 1185.343,A -85,B 0,C 180,E1 23864.111,E2 23864.111} C_VEL
LIN {X 0,Y 647.925,Z 1189.967,A -85,B 0,C 180,E1 23861.843,E2 23861.843} C_VEL
LIN {X 0,Y 647.919,Z 1193.267,A -85,B 0,C 180,E1 23859.414,E2 23859.414} C_VEL
LIN {X 0,Y 647.913,Z 1194.695,A -85,B 0,C 180,E1 23857.18,E2 23857.18} C_VEL
LIN {X 0,Y 647.906,Z 1194.821,A -85,B 0,C 180,E1 23855.224,E2 23855.224} C_VEL
LIN {X 0,Y 647.914,Z 1193.831,A -85,B 0,C 180,E1 23853.154,E2 23853.154} C_VEL
LIN {X 0,Y 647.921,Z 1191.144,A -85,B 0,C 180,E1 23850.795,E2 23850.795} C_VEL
LIN {X 0,Y 647.946,Z 1186.738,A -85,B 0,C 180,E1 23848.408,E2 23848.408} C_VEL
LIN {X 0,Y 648.02,Z 1181.153,A -85,B 0,C 180,E1 23846.195,E2 23846.195} C_VEL
LIN {X 0,Y 648.167,Z 1173.801,A -85,B 0,C 180,E1 23843.889,E2 23843.889} C_VEL
LIN {X 0,Y 648.462,Z 1163.534,A -85,B 0,C 180,E1 23841.309,E2 23841.309} C_VEL
LIN {X 0,Y 648.794,Z 1154.304,A -85,B 0,C 180,E1 23839.342,E2 23839.342} C_VEL
LIN {X 0,Y 649.245,Z 1143.727,A -85,B 0,C 180,E1 23837.368,E2 23837.368} C_VEL
LIN {X 0,Y 649.987,Z 1130.008,A -85,B 0,C 180,E1 23835.114,E2 23835.114} C_VEL
LIN {X 0,Y 650.891,Z 1114.729,A -85,B 0,C 180,E1 23832.938,E2 23832.938} C_VEL
LIN {X 0,Y 651.866,Z 1100.41,A -85,B 0,C 180,E1 23831.116,E2 23831.116} C_VEL
LIN {X 0,Y 653.226,Z 1081.91,A -85,B 0,C 180,E1 23829.011,E2 23829.011} C_VEL
LIN {X 0,Y 654.657,Z 1063.576,A -85,B 0,C 180,E1 23827.173,E2 23827.173} C_VEL
LIN {X 0,Y 656.044,Z 1046.648,A -85,B 0,C 180,E1 23825.642,E2 23825.642} C_VEL
LIN {X 0,Y 657.865,Z 1025.199,A -85,B 0,C 180,E1 23823.896,E2 23823.896} C_VEL
LIN {X 0,Y 659.646,Z 1003.042,A -85,B 0,C 180,E1 23822.316,E2 23822.316} C_VEL
LIN {X 0,Y 661.287,Z 983.287,A -85,B 0,C 180,E1 23821.063,E2 23821.063} C_VEL
LIN {X 0,Y 663.26,Z 959.427,A -85,B 0,C 180,E1 23819.722,E2 23819.722} C_VEL
LIN {X 0,Y 665.033,Z 935.069,A -85,B 0,C 180,E1 23818.552,E2 23818.552} C_VEL
LIN {X 0,Y 666.409,Z 915.013,A -85,B 0,C 180,E1 23817.714,E2 23817.714} C_VEL
LIN {X 0,Y 667.608,Z 895.151,A -85,B 0,C 180,E1 23816.989,E2 23816.989} C_VEL
LIN {X 0,Y 668.868,Z 873.28,A -85,B 0,C 180,E1 23816.31,E2 23816.31} C_VEL
LIN {X 0,Y 670.154,Z 846.986,A -85,B 0,C 180,E1 23815.65,E2 23815.65} C_VEL
LIN {X 0,Y 671.103,Z 819.906,A -85,B 0,C 180,E1 23815.15,E2 23815.15} C_VEL
LIN {X 0,Y 672.252,Z 752.981,A -85,B 0,C 180,E1 23814.268,E2 23814.268} C_VEL
LIN {X 0,Y 675.572,Z 535.127,A -85,B 0,C 180,E1 23811.416,E2 23811.416} C_VEL
LIN {X 0,Y 678.114,Z 378.482,A -85,B 0,C 180,E1 23809.309,E2 23809.309} C_VEL
LIN {X 0,Y 663.745,Z 357.208,A -85,B 0,C 180,E1 23807.639,E2 23807.639} C_VEL
LIN {X 0,Y 655.597,Z 345.994,A -85,B 0,C 180,E1 23806.646,E2 23806.646} C_VEL
LIN {X 0,Y 652.035,Z 340.987,A -85,B 0,C 180,E1 23806.179,E2 23806.179} C_VEL
LIN {X 0,Y 650.262,Z 337.174,A -85,B 0,C 180,E1 23805.645,E2 23805.645} C_VEL
LIN {X 0,Y 648.927,Z 334.323,A -85,B 0,C 180,E1 23805.239,E2 23805.239} C_VEL
LIN {X 0,Y 648.766,Z 333.422,A -85,B 0,C 180,E1 23805.1,E2 23805.1} C_VEL
LIN {X 0,Y 648.744,Z 333.419,A -85,B 0,C 180,E1 23802.022,E2 23802.022} C_VEL
LIN {X 0,Y 648.773,Z 333.422,A -85,B 0,C 180,E1 23798.849,E2 23798.849} C_VEL
LIN {X 0,Y 648.747,Z 333.416,A -85,B 0,C 180,E1 23795.742,E2 23795.742} C_VEL
LIN {X 0,Y 648.75,Z 333.42,A -85,B 0,C 180,E1 23792.535,E2 23792.535} C_VEL
LIN {X 0,Y 648.745,Z 333.416,A -85,B 0,C 180,E1 23789.552,E2 23789.552} C_VEL
LIN {X 0,Y 648.736,Z 333.389,A -85,B 0,C 180,E1 23786.353,E2 23786.353} C_VEL
LIN {X 0,Y 648.739,Z 333.417,A -85,B 0,C 180,E1 23783.432,E2 23783.432} C_VEL
LIN {X 0,Y 648.725,Z 333.389,A -85,B 0,C 180,E1 23780.197,E2 23780.197} C_VEL
LIN {X 0,Y 648.733,Z 333.417,A -85,B 0,C 180,E1 23777.306,E2 23777.306} C_VEL
LIN {X 0,Y 648.722,Z 333.384,A -85,B 0,C 180,E1 23774.095,E2 23774.095} C_VEL
LIN {X 0,Y 648.715,Z 333.415,A -85,B 0,C 180,E1 23771.289,E2 23771.289} C_VEL
LIN {X 0,Y 648.739,Z 333.417,A -85,B 0,C 180,E1 23768.152,E2 23768.152} C_VEL
LIN {X 0,Y 648.697,Z 333.414,A -85,B 0,C 180,E1 23765.395,E2 23765.395} C_VEL
LIN {X 0,Y 648.77,Z 333.415,A -85,B 0,C 180,E1 23762.385,E2 23762.385} C_VEL
LIN {X 0,Y 648.692,Z 333.422,A -85,B 0,C 180,E1 23759.47,E2 23759.47} C_VEL
LIN {X 0,Y 648.719,Z 333.419,A -85,B 0,C 180,E1 23756.731,E2 23756.731} C_VEL
LIN {X 0,Y 648.7,Z 333.425,A -85,B 0,C 180,E1 23753.628,E2 23753.628} C_VEL
LIN {X 0,Y 648.68,Z 333.416,A -85,B 0,C 180,E1 23751.044,E2 23751.044} C_VEL
LIN {X 0,Y 648.76,Z 333.404,A -85,B 0,C 180,E1 23748.081,E2 23748.081} C_VEL
LIN {X 0,Y 648.673,Z 333.412,A -85,B 0,C 180,E1 23745.174,E2 23745.174} C_VEL
LIN {X 0,Y 648.686,Z 333.425,A -85,B 0,C 180,E1 23742.577,E2 23742.577} C_VEL
LIN {X 0,Y 648.681,Z 333.407,A -85,B 0,C 180,E1 23739.33,E2 23739.33} C_VEL
LIN {X 0,Y 648.662,Z 333.425,A -85,B 0,C 180,E1 23736.758,E2 23736.758} C_VEL
LIN {X 0,Y 648.743,Z 333.394,A -85,B 0,C 180,E1 23733.845,E2 23733.845} C_VEL
LIN {X 0,Y 648.671,Z 333.422,A -85,B 0,C 180,E1 23730.926,E2 23730.926} C_VEL
LIN {X 0,Y 648.68,Z 333.42,A -85,B 0,C 180,E1 23728.393,E2 23728.393} C_VEL
LIN {X 0,Y 648.731,Z 333.424,A -85,B 0,C 180,E1 23725.337,E2 23725.337} C_VEL
LIN {X 0,Y 648.68,Z 333.43,A -85,B 0,C 180,E1 23722.544,E2 23722.544} C_VEL
LIN {X 0,Y 648.766,Z 333.457,A -85,B 0,C 180,E1 23721.602,E2 23721.602} C_VEL
LIN {X 0,Y 650.115,Z 337.037,A -85,B 0,C 180,E1 23721.133,E2 23721.133} C_VEL
LIN {X 0,Y 651.097,Z 339,A -85,B 0,C 180,E1 23720.852,E2 23720.852} C_VEL
LIN {X 0,Y 657.012,Z 350.863,A -85,B 0,C 180,E1 23719.24,E2 23719.24} C_VEL
LIN {X 0,Y 674.776,Z 376.529,A -85,B 0,C 180,E1 23717.13,E2 23717.13} C_VEL
LIN {X 0,Y 678.257,Z 382.059,A -85,B 0,C 180,E1 23716.73,E2 23716.73} C_VEL
LIN {X 0,Y 674.841,Z 592.238,A -85,B 0,C 180,E1 23713.914,E2 23713.914} C_VEL
LIN {X 0,Y 671.495,Z 815.177,A -85,B 0,C 180,E1 23711.016,E2 23711.016} C_VEL
LIN {X 0,Y 670.676,Z 842.649,A -85,B 0,C 180,E1 23710.588,E2 23710.588} C_VEL
LIN {X 0,Y 669.718,Z 866.02,A -85,B 0,C 180,E1 23710.094,E2 23710.094} C_VEL
LIN {X 0,Y 668.455,Z 891.547,A -85,B 0,C 180,E1 23709.407,E2 23709.407} C_VEL
LIN {X 0,Y 666.805,Z 918.723,A -85,B 0,C 180,E1 23708.484,E2 23708.484} C_VEL
LIN {X 0,Y 665.362,Z 939.925,A -85,B 0,C 180,E1 23707.63,E2 23707.63} C_VEL
LIN {X 0,Y 663.855,Z 960.701,A -85,B 0,C 180,E1 23706.67,E2 23706.67} C_VEL
LIN {X 0,Y 662.099,Z 983.891,A -85,B 0,C 180,E1 23705.444,E2 23705.444} C_VEL
LIN {X 0,Y 660.057,Z 1008.591,A -85,B 0,C 180,E1 23703.933,E2 23703.933} C_VEL
LIN {X 0,Y 658.451,Z 1027.569,A -85,B 0,C 180,E1 23702.621,E2 23702.621} C_VEL
LIN {X 0,Y 656.824,Z 1047.075,A -85,B 0,C 180,E1 23701.119,E2 23701.119} C_VEL
LIN {X 0,Y 654.985,Z 1069.749,A -85,B 0,C 180,E1 23699.142,E2 23699.142} C_VEL
LIN {X 0,Y 653.646,Z 1086.381,A -85,B 0,C 180,E1 23697.514,E2 23697.514} C_VEL
LIN {X 0,Y 652.371,Z 1103.303,A -85,B 0,C 180,E1 23695.679,E2 23695.679} C_VEL
LIN {X 0,Y 651.105,Z 1121.56,A -85,B 0,C 180,E1 23693.437,E2 23693.437} C_VEL
LIN {X 0,Y 650.245,Z 1135.429,A -85,B 0,C 180,E1 23691.515,E2 23691.515} C_VEL
LIN {X 0,Y 649.487,Z 1149.549,A -85,B 0,C 180,E1 23689.313,E2 23689.313} C_VEL
LIN {X 0,Y 648.875,Z 1162.211,A -85,B 0,C 180,E1 23687.025,E2 23687.025} C_VEL
LIN {X 0,Y 648.513,Z 1171.484,A -85,B 0,C 180,E1 23685.104,E2 23685.104} C_VEL
LIN {X 0,Y 648.279,Z 1179.513,A -85,B 0,C 180,E1 23683.195,E2 23683.195} C_VEL
LIN {X 0,Y 648.084,Z 1187.034,A -85,B 0,C 180,E1 23681.112,E2 23681.112} C_VEL
LIN {X 0,Y 647.987,Z 1194.034,A -85,B 0,C 180,E1 23678.698,E2 23678.698} C_VEL
LIN {X 0,Y 647.935,Z 1199.101,A -85,B 0,C 180,E1 23676.372,E2 23676.372} C_VEL
LIN {X 0,Y 647.918,Z 1202.476,A -85,B 0,C 180,E1 23674.16,E2 23674.16} C_VEL
LIN {X 0,Y 647.908,Z 1204.549,A -85,B 0,C 180,E1 23671.769,E2 23671.769} C_VEL
LIN {X 0,Y 647.892,Z 1204.872,A -85,B 0,C 180,E1 23669.47,E2 23669.47} C_VEL
LIN {X 0,Y 647.91,Z 1203.944,A -85,B 0,C 180,E1 23667.347,E2 23667.347} C_VEL
LIN {X 0,Y 647.922,Z 1201.428,A -85,B 0,C 180,E1 23665.043,E2 23665.043} C_VEL
LIN {X 0,Y 647.951,Z 1197.152,A -85,B 0,C 180,E1 23662.642,E2 23662.642} C_VEL
LIN {X 0,Y 648.018,Z 1191.373,A -85,B 0,C 180,E1 23660.318,E2 23660.318} C_VEL
LIN {X 0,Y 648.146,Z 1184.279,A -85,B 0,C 180,E1 23658.07,E2 23658.07} C_VEL
LIN {X 0,Y 648.44,Z 1174.338,A -85,B 0,C 180,E1 23655.535,E2 23655.535} C_VEL
LIN {X 0,Y 648.771,Z 1164.544,A -85,B 0,C 180,E1 23653.434,E2 23653.434} C_VEL
LIN {X 0,Y 649.238,Z 1154.237,A -85,B 0,C 180,E1 23651.503,E2 23651.503} C_VEL
LIN {X 0,Y 649.924,Z 1141.364,A -85,B 0,C 180,E1 23649.372,E2 23649.372} C_VEL
LIN {X 0,Y 650.838,Z 1125.802,A -85,B 0,C 180,E1 23647.128,E2 23647.128} C_VEL
LIN {X 0,Y 651.804,Z 1111.151,A -85,B 0,C 180,E1 23645.251,E2 23645.251} C_VEL
LIN {X 0,Y 653.113,Z 1093.726,A -85,B 0,C 180,E1 23643.251,E2 23643.251} C_VEL
LIN {X 0,Y 654.549,Z 1074.83,A -85,B 0,C 180,E1 23641.337,E2 23641.337} C_VEL
LIN {X 0,Y 655.938,Z 1057.949,A -85,B 0,C 180,E1 23639.8,E2 23639.8} C_VEL
LIN {X 0,Y 657.512,Z 1039.191,A -85,B 0,C 180,E1 23638.254,E2 23638.254} C_VEL
LIN {X 0,Y 659.487,Z 1015.131,A -85,B 0,C 180,E1 23636.501,E2 23636.501} C_VEL
LIN {X 0,Y 661.14,Z 994.955,A -85,B 0,C 180,E1 23635.207,E2 23635.207} C_VEL
LIN {X 0,Y 662.831,Z 974.056,A -85,B 0,C 180,E1 23634.017,E2 23634.017} C_VEL
LIN {X 0,Y 664.822,Z 948.469,A -85,B 0,C 180,E1 23632.746,E2 23632.746} C_VEL
LIN {X 0,Y 666.407,Z 925.166,A -85,B 0,C 180,E1 23631.764,E2 23631.764} C_VEL
LIN {X 0,Y 667.662,Z 904.462,A -85,B 0,C 180,E1 23631.01,E2 23631.01} C_VEL
LIN {X 0,Y 668.912,Z 882.296,A -85,B 0,C 180,E1 23630.327,E2 23630.327} C_VEL
LIN {X 0,Y 670.162,Z 856.667,A -85,B 0,C 180,E1 23629.689,E2 23629.689} C_VEL
LIN {X 0,Y 671.133,Z 829.097,A -85,B 0,C 180,E1 23629.182,E2 23629.182} C_VEL
LIN {X 0,Y 673.011,Z 711.796,A -85,B 0,C 180,E1 23627.65,E2 23627.65} C_VEL
LIN {X 0,Y 676.421,Z 493.199,A -85,B 0,C 180,E1 23624.77,E2 23624.77} C_VEL
LIN {X 0,Y 678.143,Z 381.615,A -85,B 0,C 180,E1 23623.253,E2 23623.253} C_VEL
LIN {X 0,Y 663.414,Z 359.987,A -85,B 0,C 180,E1 23621.542,E2 23621.542} C_VEL
LIN {X 0,Y 656.499,Z 350.035,A -85,B 0,C 180,E1 23620.671,E2 23620.671} C_VEL
LIN {X 0,Y 652.316,Z 341.515,A -85,B 0,C 180,E1 23619.504,E2 23619.504} C_VEL
LIN {X 0,Y 650.101,Z 337.016,A -85,B 0,C 180,E1 23618.868,E2 23618.868} C_VEL
LIN {X 0,Y 648.761,Z 333.42,A -85,B 0,C 180,E1 23618.363,E2 23618.363} C_VEL
LIN {X 0,Y 648.682,Z 333.42,A -85,B 0,C 180,E1 23615.526,E2 23615.526} C_VEL
LIN {X 0,Y 648.703,Z 333.423,A -85,B 0,C 180,E1 23612.857,E2 23612.857} C_VEL
LIN {X 0,Y 648.69,Z 333.413,A -85,B 0,C 180,E1 23609.656,E2 23609.656} C_VEL
LIN {X 0,Y 648.672,Z 333.413,A -85,B 0,C 180,E1 23607.147,E2 23607.147} C_VEL
LIN {X 0,Y 648.756,Z 333.42,A -85,B 0,C 180,E1 23604.162,E2 23604.162} C_VEL
LIN {X 0,Y 648.668,Z 333.405,A -85,B 0,C 180,E1 23601.238,E2 23601.238} C_VEL
LIN {X 0,Y 648.68,Z 333.427,A -85,B 0,C 180,E1 23598.607,E2 23598.607} C_VEL
LIN {X 0,Y 648.681,Z 333.417,A -85,B 0,C 180,E1 23595.374,E2 23595.374} C_VEL
LIN {X 0,Y 648.662,Z 333.422,A -85,B 0,C 180,E1 23592.825,E2 23592.825} C_VEL
LIN {X 0,Y 648.737,Z 333.406,A -85,B 0,C 180,E1 23589.94,E2 23589.94} C_VEL
LIN {X 0,Y 648.673,Z 333.412,A -85,B 0,C 180,E1 23586.945,E2 23586.945} C_VEL
LIN {X 0,Y 648.682,Z 333.414,A -85,B 0,C 180,E1 23584.332,E2 23584.332} C_VEL
LIN {X 0,Y 648.715,Z 333.401,A -85,B 0,C 180,E1 23581.236,E2 23581.236} C_VEL
LIN {X 0,Y 648.677,Z 333.42,A -85,B 0,C 180,E1 23578.587,E2 23578.587} C_VEL
LIN {X 0,Y 648.717,Z 333.407,A -85,B 0,C 180,E1 23575.846,E2 23575.846} C_VEL
LIN {X 0,Y 648.695,Z 333.423,A -85,B 0,C 180,E1 23572.739,E2 23572.739} C_VEL
LIN {X 0,Y 648.686,Z 333.408,A -85,B 0,C 180,E1 23570.148,E2 23570.148} C_VEL
LIN {X 0,Y 648.757,Z 333.42,A -85,B 0,C 180,E1 23567.086,E2 23567.086} C_VEL
LIN {X 0,Y 648.687,Z 333.394,A -85,B 0,C 180,E1 23564.259,E2 23564.259} C_VEL
LIN {X 0,Y 648.745,Z 333.418,A -85,B 0,C 180,E1 23561.416,E2 23561.416} C_VEL
LIN {X 0,Y 648.703,Z 333.42,A -85,B 0,C 180,E1 23558.345,E2 23558.345} C_VEL
LIN {X 0,Y 648.706,Z 333.405,A -85,B 0,C 180,E1 23555.698,E2 23555.698} C_VEL
LIN {X 0,Y 648.743,Z 333.415,A -85,B 0,C 180,E1 23552.558,E2 23552.558} C_VEL
LIN {X 0,Y 648.705,Z 333.42,A -85,B 0,C 180,E1 23549.733,E2 23549.733} C_VEL
LIN {X 0,Y 648.802,Z 333.618,A -85,B 0,C 180,E1 23546.755,E2 23546.755} C_VEL
LIN {X 0,Y 650.203,Z 337.142,A -85,B 0,C 180,E1 23546.279,E2 23546.279} C_VEL
LIN {X 0,Y 652.551,Z 341.742,A -85,B 0,C 180,E1 23545.649,E2 23545.649} C_VEL
LIN {X 0,Y 658.132,Z 349.547,A -85,B 0,C 180,E1 23544.95,E2 23544.95} C_VEL
LIN {X 0,Y 669.682,Z 365.852,A -85,B 0,C 180,E1 23543.567,E2 23543.567} C_VEL
LIN {X 0,Y 678.173,Z 378.781,A -85,B 0,C 180,E1 23542.591,E2 23542.591} C_VEL
LIN {X 0,Y 677.826,Z 399.518,A -85,B 0,C 180,E1 23542.309,E2 23542.309} C_VEL
LIN {X 0,Y 677.002,Z 407.224,A -85,B 0,C 180,E1 23542.267,E2 23542.267} C_VEL
LIN {X 0,Y 672.29,Z 427.908,A -85,B 0,C 180,E1 23542.374,E2 23542.374} C_VEL
LIN {X 0,Y 671.657,Z 434.517,A -85,B 0,C 180,E1 23542.33,E2 23542.33} C_VEL
LIN {X 0,Y 667.951,Z 649.304,A -85,B 0,C 180,E1 23539.459,E2 23539.459} C_VEL
LIN {X 0,Y 665.098,Z 817.831,A -85,B 0,C 180,E1 23537.243,E2 23537.243} C_VEL
LIN {X 0,Y 664.187,Z 843.179,A -85,B 0,C 180,E1 23536.79,E2 23536.79} C_VEL
LIN {X 0,Y 662.776,Z 871.008,A -85,B 0,C 180,E1 23536.112,E2 23536.112} C_VEL
LIN {X 0,Y 661.446,Z 893.095,A -85,B 0,C 180,E1 23535.433,E2 23535.433} C_VEL
LIN {X 0,Y 660.177,Z 912.405,A -85,B 0,C 180,E1 23534.737,E2 23534.737} C_VEL
LIN {X 0,Y 658.715,Z 932.158,A -85,B 0,C 180,E1 23533.922,E2 23533.922} C_VEL
LIN {X 0,Y 657.052,Z 953.366,A -85,B 0,C 180,E1 23532.92,E2 23532.92} C_VEL
LIN {X 0,Y 654.972,Z 978.405,A -85,B 0,C 180,E1 23531.558,E2 23531.558} C_VEL
LIN {X 0,Y 653.091,Z 999.326,A -85,B 0,C 180,E1 23530.246,E2 23530.246} C_VEL
LIN {X 0,Y 651.395,Z 1017.93,A -85,B 0,C 180,E1 23528.944,E2 23528.944} C_VEL
LIN {X 0,Y 649.699,Z 1036.611,A -85,B 0,C 180,E1 23527.493,E2 23527.493} C_VEL
LIN {X 0,Y 647.766,Z 1058.676,A -85,B 0,C 180,E1 23525.563,E2 23525.563} C_VEL
LIN {X 0,Y 646.215,Z 1076.436,A -85,B 0,C 180,E1 23523.808,E2 23523.808} C_VEL
LIN {X 0,Y 644.827,Z 1093.072,A -85,B 0,C 180,E1 23521.983,E2 23521.983} C_VEL
LIN {X 0,Y 643.449,Z 1111.364,A -85,B 0,C 180,E1 23519.716,E2 23519.716} C_VEL
LIN {X 0,Y 642.483,Z 1125.516,A -85,B 0,C 180,E1 23517.731,E2 23517.731} C_VEL
LIN {X 0,Y 641.639,Z 1139.793,A -85,B 0,C 180,E1 23515.473,E2 23515.473} C_VEL
LIN {X 0,Y 640.964,Z 1152.461,A -85,B 0,C 180,E1 23513.148,E2 23513.148} C_VEL
LIN {X 0,Y 640.572,Z 1162.003,A -85,B 0,C 180,E1 23511.135,E2 23511.135} C_VEL
LIN {X 0,Y 640.291,Z 1170.245,A -85,B 0,C 180,E1 23509.129,E2 23509.129} C_VEL
LIN {X 0,Y 640.089,Z 1178.354,A -85,B 0,C 180,E1 23506.797,E2 23506.797} C_VEL
LIN {X 0,Y 639.981,Z 1184.965,A -85,B 0,C 180,E1 23504.378,E2 23504.378} C_VEL
LIN {X 0,Y 639.928,Z 1189.667,A -85,B 0,C 180,E1 23502.085,E2 23502.085} C_VEL
LIN {X 0,Y 639.912,Z 1192.995,A -85,B 0,C 180,E1 23499.715,E2 23499.715} C_VEL
LIN {X 0,Y 639.913,Z 1194.653,A -85,B 0,C 180,E1 23497.361,E2 23497.361} C_VEL
LIN {X 0,Y 639.903,Z 1194.84,A -85,B 0,C 180,E1 23495.289,E2 23495.289} C_VEL
LIN {X 0,Y 639.911,Z 1193.909,A -85,B 0,C 180,E1 23493.224,E2 23493.224} C_VEL
LIN {X 0,Y 639.922,Z 1191.373,A -85,B 0,C 180,E1 23490.895,E2 23490.895} C_VEL
LIN {X 0,Y 639.949,Z 1187.094,A -85,B 0,C 180,E1 23488.478,E2 23488.478} C_VEL
LIN {X 0,Y 640.029,Z 1181.361,A -85,B 0,C 180,E1 23486.148,E2 23486.148} C_VEL
LIN {X 0,Y 640.19,Z 1174.067,A -85,B 0,C 180,E1 23483.813,E2 23483.813} C_VEL
LIN {X 0,Y 640.505,Z 1163.87,A -85,B 0,C 180,E1 23481.2,E2 23481.2} C_VEL
LIN {X 0,Y 640.896,Z 1154.24,A -85,B 0,C 180,E1 23479.118,E2 23479.118} C_VEL
LIN {X 0,Y 641.411,Z 1143.657,A -85,B 0,C 180,E1 23477.119,E2 23477.119} C_VEL
LIN {X 0,Y 642.24,Z 1129.309,A -85,B 0,C 180,E1 23474.745,E2 23474.745} C_VEL
LIN {X 0,Y 643.201,Z 1114.637,A -85,B 0,C 180,E1 23472.634,E2 23472.634} C_VEL
LIN {X 0,Y 644.349,Z 1099.56,A -85,B 0,C 180,E1 23470.699,E2 23470.699} C_VEL
LIN {X 0,Y 645.888,Z 1080.02,A -85,B 0,C 180,E1 23468.476,E2 23468.476} C_VEL
LIN {X 0,Y 647.342,Z 1063.278,A -85,B 0,C 180,E1 23466.787,E2 23466.787} C_VEL
LIN {X 0,Y 648.858,Z 1046.097,A -85,B 0,C 180,E1 23465.219,E2 23465.219} C_VEL
LIN {X 0,Y 650.824,Z 1024.405,A -85,B 0,C 180,E1 23463.444,E2 23463.444} C_VEL
LIN {X 0,Y 652.705,Z 1003.344,A -85,B 0,C 180,E1 23461.932,E2 23461.932} C_VEL
LIN {X 0,Y 654.448,Z 983.841,A -85,B 0,C 180,E1 23460.681,E2 23460.681} C_VEL
LIN {X 0,Y 656.4,Z 961.656,A -85,B 0,C 180,E1 23459.418,E2 23459.418} C_VEL
LIN {X 0,Y 658.468,Z 935.819,A -85,B 0,C 180,E1 23458.151,E2 23458.151} C_VEL
LIN {X 0,Y 660.028,Z 914.647,A -85,B 0,C 180,E1 23457.26,E2 23457.26} C_VEL
LIN {X 0,Y 661.325,Z 894.744,A -85,B 0,C 180,E1 23456.531,E2 23456.531} C_VEL
LIN {X 0,Y 662.663,Z 872.95,A -85,B 0,C 180,E1 23455.854,E2 23455.854} C_VEL
LIN {X 0,Y 664.045,Z 846.633,A -85,B 0,C 180,E1 23455.193,E2 23455.193} C_VEL
LIN {X 0,Y 665.042,Z 819.813,A -85,B 0,C 180,E1 23454.697,E2 23454.697} C_VEL
LIN {X 0,Y 666.24,Z 755.151,A -85,B 0,C 180,E1 23453.837,E2 23453.837} C_VEL
LIN {X 0,Y 669.841,Z 536.603,A -85,B 0,C 180,E1 23450.954,E2 23450.954} C_VEL
LIN {X 0,Y 672.504,Z 382.206,A -85,B 0,C 180,E1 23448.858,E2 23448.858} C_VEL
LIN {X 0,Y 659.294,Z 362.7,A -85,B 0,C 180,E1 23447.29,E2 23447.29} C_VEL
LIN {X 0,Y 648.328,Z 347.426,A -85,B 0,C 180,E1 23445.915,E2 23445.915} C_VEL
LIN {X 0,Y 643.616,Z 340.975,A -85,B 0,C 180,E1 23445.271,E2 23445.271} C_VEL
LIN {X 0,Y 642.6,Z 338.52,A -85,B 0,C 180,E1 23444.929,E2 23444.929} C_VEL
LIN {X 0,Y 640.995,Z 335.424,A -85,B 0,C 180,E1 23444.459,E2 23444.459} C_VEL
LIN {X 0,Y 640.801,Z 334.412,A -85,B 0,C 180,E1 23444.33,E2 23444.33} C_VEL
LIN {X 0,Y 640.825,Z 334.404,A -85,B 0,C 180,E1 23441.23,E2 23441.23} C_VEL
LIN {X 0,Y 640.795,Z 334.408,A -85,B 0,C 180,E1 23438.278,E2 23438.278} C_VEL
LIN {X 0,Y 640.829,Z 334.402,A -85,B 0,C 180,E1 23435.262,E2 23435.262} C_VEL
LIN {X 0,Y 640.791,Z 334.411,A -85,B 0,C 180,E1 23432.147,E2 23432.147} C_VEL
LIN {X 0,Y 640.834,Z 334.406,A -85,B 0,C 180,E1 23429.102,E2 23429.102} C_VEL
LIN {X 0,Y 640.783,Z 334.379,A -85,B 0,C 180,E1 23426.107,E2 23426.107} C_VEL
LIN {X 0,Y 640.832,Z 334.406,A -85,B 0,C 180,E1 23423.056,E2 23423.056} C_VEL
LIN {X 0,Y 640.775,Z 334.377,A -85,B 0,C 180,E1 23419.983,E2 23419.983} C_VEL
LIN {X 0,Y 640.818,Z 334.405,A -85,B 0,C 180,E1 23417.058,E2 23417.058} C_VEL
LIN {X 0,Y 640.772,Z 334.371,A -85,B 0,C 180,E1 23413.905,E2 23413.905} C_VEL
LIN {X 0,Y 640.797,Z 334.403,A -85,B 0,C 180,E1 23411.047,E2 23411.047} C_VEL
LIN {X 0,Y 640.775,Z 334.412,A -85,B 0,C 180,E1 23407.893,E2 23407.893} C_VEL
LIN {X 0,Y 640.766,Z 334.402,A -85,B 0,C 180,E1 23405.193,E2 23405.193} C_VEL
LIN {X 0,Y 640.796,Z 334.403,A -85,B 0,C 180,E1 23402.057,E2 23402.057} C_VEL
LIN {X 0,Y 640.753,Z 334.41,A -85,B 0,C 180,E1 23399.285,E2 23399.285} C_VEL
LIN {X 0,Y 640.825,Z 334.409,A -85,B 0,C 180,E1 23396.332,E2 23396.332} C_VEL
LIN {X 0,Y 640.748,Z 334.413,A -85,B 0,C 180,E1 23393.369,E2 23393.369} C_VEL
LIN {X 0,Y 640.757,Z 334.404,A -85,B 0,C 180,E1 23390.751,E2 23390.751} C_VEL
LIN {X 0,Y 640.757,Z 334.389,A -85,B 0,C 180,E1 23387.564,E2 23387.564} C_VEL
LIN {X 0,Y 640.735,Z 334.403,A -85,B 0,C 180,E1 23384.894,E2 23384.894} C_VEL
LIN {X 0,Y 640.811,Z 334.393,A -85,B 0,C 180,E1 23381.91,E2 23381.91} C_VEL
LIN {X 0,Y 640.726,Z 334.406,A -85,B 0,C 180,E1 23378.94,E2 23378.94} C_VEL
LIN {X 0,Y 640.757,Z 334.403,A -85,B 0,C 180,E1 23376.259,E2 23376.259} C_VEL
LIN {X 0,Y 640.738,Z 334.412,A -85,B 0,C 180,E1 23373.092,E2 23373.092} C_VEL
LIN {X 0,Y 640.737,Z 334.412,A -85,B 0,C 180,E1 23370.453,E2 23370.453} C_VEL
LIN {X 0,Y 640.796,Z 334.412,A -85,B 0,C 180,E1 23367.416,E2 23367.416} C_VEL
LIN {X 0,Y 640.739,Z 334.418,A -85,B 0,C 180,E1 23364.547,E2 23364.547} C_VEL
LIN {X 0,Y 640.746,Z 334.438,A -85,B 0,C 180,E1 23362.399,E2 23362.399} C_VEL
LIN {X 0,Y 642.106,Z 337.934,A -85,B 0,C 180,E1 23361.928,E2 23361.928} C_VEL
LIN {X 0,Y 643.147,Z 339.612,A -85,B 0,C 180,E1 23361.66,E2 23361.66} C_VEL
LIN {X 0,Y 648.591,Z 350.82,A -85,B 0,C 180,E1 23360.109,E2 23360.109} C_VEL
LIN {X 0,Y 662.821,Z 370.98,A -85,B 0,C 180,E1 23358.34,E2 23358.34} C_VEL
LIN {X 0,Y 672.699,Z 385.795,A -85,B 0,C 180,E1 23357.178,E2 23357.178} C_VEL
LIN {X 0,Y 669.03,Z 594.927,A -85,B 0,C 180,E1 23354.356,E2 23354.356} C_VEL
LIN {X 0,Y 665.384,Z 818.172,A -85,B 0,C 180,E1 23351.429,E2 23351.429} C_VEL
LIN {X 0,Y 664.542,Z 843.598,A -85,B 0,C 180,E1 23351.022,E2 23351.022} C_VEL
LIN {X 0,Y 663.521,Z 866.781,A -85,B 0,C 180,E1 23350.524,E2 23350.524} C_VEL
LIN {X 0,Y 662.121,Z 893.014,A -85,B 0,C 180,E1 23349.809,E2 23349.809} C_VEL
LIN {X 0,Y 660.372,Z 919.444,A -85,B 0,C 180,E1 23348.898,E2 23348.898} C_VEL
LIN {X 0,Y 658.812,Z 940.777,A -85,B 0,C 180,E1 23348.029,E2 23348.029} C_VEL
LIN {X 0,Y 657.098,Z 962.801,A -85,B 0,C 180,E1 23346.995,E2 23346.995} C_VEL
LIN {X 0,Y 654.915,Z 988.946,A -85,B 0,C 180,E1 23345.569,E2 23345.569} C_VEL
LIN {X 0,Y 652.995,Z 1010.38,A -85,B 0,C 180,E1 23344.221,E2 23344.221} C_VEL
LIN {X 0,Y 651.255,Z 1029.467,A -85,B 0,C 180,E1 23342.878,E2 23342.878} C_VEL
LIN {X 0,Y 649.323,Z 1051.28,A -85,B 0,C 180,E1 23341.158,E2 23341.158} C_VEL
LIN {X 0,Y 647.52,Z 1071.272,A -85,B 0,C 180,E1 23339.359,E2 23339.359} C_VEL
LIN {X 0,Y 646.095,Z 1087.7,A -85,B 0,C 180,E1 23337.721,E2 23337.721} C_VEL
LIN {X 0,Y 644.596,Z 1106.396,A -85,B 0,C 180,E1 23335.644,E2 23335.644} C_VEL
LIN {X 0,Y 643.325,Z 1122.983,A -85,B 0,C 180,E1 23333.543,E2 23333.543} C_VEL
LIN {X 0,Y 642.422,Z 1136.379,A -85,B 0,C 180,E1 23331.646,E2 23331.646} C_VEL
LIN {X 0,Y 641.56,Z 1151.096,A -85,B 0,C 180,E1 23329.294,E2 23329.294} C_VEL
LIN {X 0,Y 640.933,Z 1163.143,A -85,B 0,C 180,E1 23327.055,E2 23327.055} C_VEL
LIN {X 0,Y 640.55,Z 1172.307,A -85,B 0,C 180,E1 23325.111,E2 23325.111} C_VEL
LIN {X 0,Y 640.289,Z 1180.576,A -85,B 0,C 180,E1 23323.087,E2 23323.087} C_VEL
LIN {X 0,Y 640.074,Z 1188.477,A -85,B 0,C 180,E1 23320.805,E2 23320.805} C_VEL
LIN {X 0,Y 639.978,Z 1195.119,A -85,B 0,C 180,E1 23318.355,E2 23318.355} C_VEL
LIN {X 0,Y 639.931,Z 1199.723,A -85,B 0,C 180,E1 23316.099,E2 23316.099} C_VEL
LIN {X 0,Y 639.912,Z 1203.094,A -85,B 0,C 180,E1 23313.673,E2 23313.673} C_VEL
LIN {X 0,Y 639.914,Z 1204.669,A -85,B 0,C 180,E1 23311.343,E2 23311.343} C_VEL
LIN {X 0,Y 639.894,Z 1204.849,A -85,B 0,C 180,E1 23309.374,E2 23309.374} C_VEL
LIN {X 0,Y 639.911,Z 1203.942,A -85,B 0,C 180,E1 23307.314,E2 23307.314} C_VEL
LIN {X 0,Y 639.922,Z 1201.553,A -85,B 0,C 180,E1 23305.07,E2 23305.07} C_VEL
LIN {X 0,Y 639.953,Z 1197.347,A -85,B 0,C 180,E1 23302.639,E2 23302.639} C_VEL
LIN {X 0,Y 640.026,Z 1191.625,A -85,B 0,C 180,E1 23300.287,E2 23300.287} C_VEL
LIN {X 0,Y 640.164,Z 1184.591,A -85,B 0,C 180,E1 23298.011,E2 23298.011} C_VEL
LIN {X 0,Y 640.484,Z 1174.742,A -85,B 0,C 180,E1 23295.444,E2 23295.444} C_VEL
LIN {X 0,Y 640.843,Z 1165.002,A -85,B 0,C 180,E1 23293.317,E2 23293.317} C_VEL
LIN {X 0,Y 641.35,Z 1154.761,A -85,B 0,C 180,E1 23291.362,E2 23291.362} C_VEL
LIN {X 0,Y 642.053,Z 1142.531,A -85,B 0,C 180,E1 23289.298,E2 23289.298} C_VEL
LIN {X 0,Y 643.082,Z 1126.501,A -85,B 0,C 180,E1 23286.933,E2 23286.933} C_VEL
LIN {X 0,Y 644.144,Z 1111.858,A -85,B 0,C 180,E1 23285.026,E2 23285.026} C_VEL
LIN {X 0,Y 645.467,Z 1095.434,A -85,B 0,C 180,E1 23283.107,E2 23283.107} C_VEL
LIN {X 0,Y 647.157,Z 1075.335,A -85,B 0,C 180,E1 23281.03,E2 23281.03} C_VEL
LIN {X 0,Y 648.611,Z 1058.94,A -85,B 0,C 180,E1 23279.514,E2 23279.514} C_VEL
LIN {X 0,Y 650.171,Z 1041.623,A -85,B 0,C 180,E1 23278.061,E2 23278.061} C_VEL
LIN {X 0,Y 652.2,Z 1019.546,A -85,B 0,C 180,E1 23276.397,E2 23276.397} C_VEL
LIN {X 0,Y 654.205,Z 996.472,A -85,B 0,C 180,E1 23274.885,E2 23274.885} C_VEL
LIN {X 0,Y 655.998,Z 975.852,A -85,B 0,C 180,E1 23273.691,E2 23273.691} C_VEL
LIN {X 0,Y 657.99,Z 952.259,A -85,B 0,C 180,E1 23272.49,E2 23272.49} C_VEL
LIN {X 0,Y 659.917,Z 926.442,A -85,B 0,C 180,E1 23271.374,E2 23271.374} C_VEL
LIN {X 0,Y 661.329,Z 904.866,A -85,B 0,C 180,E1 23270.58,E2 23270.58} C_VEL
LIN {X 0,Y 662.657,Z 882.906,A -85,B 0,C 180,E1 23269.898,E2 23269.898} C_VEL
LIN {X 0,Y 663.967,Z 857.915,A -85,B 0,C 180,E1 23269.267,E2 23269.267} C_VEL
LIN {X 0,Y 665.054,Z 829.721,A -85,B 0,C 180,E1 23268.74,E2 23268.74} C_VEL
LIN {X 0,Y 666.547,Z 746.278,A -85,B 0,C 180,E1 23267.636,E2 23267.636} C_VEL
LIN {X 0,Y 670.263,Z 523.482,A -85,B 0,C 180,E1 23264.691,E2 23264.691} C_VEL
LIN {X 0,Y 672.614,Z 385.44,A -85,B 0,C 180,E1 23262.809,E2 23262.809} C_VEL
LIN {X 0,Y 656.333,Z 361.652,A -85,B 0,C 180,E1 23260.869,E2 23260.869} C_VEL
LIN {X 0,Y 648.008,Z 349.883,A -85,B 0,C 180,E1 23259.789,E2 23259.789} C_VEL
LIN {X 0,Y 643.988,Z 341.709,A -85,B 0,C 180,E1 23258.621,E2 23258.621} C_VEL
LIN {X 0,Y 642.532,Z 338.478,A -85,B 0,C 180,E1 23258.156,E2 23258.156} C_VEL
LIN {X 0,Y 640.978,Z 335.553,A -85,B 0,C 180,E1 23257.698,E2 23257.698} C_VEL
LIN {X 0,Y 640.747,Z 334.415,A -85,B 0,C 180,E1 23257.56,E2 23257.56} C_VEL
LIN {X 0,Y 640.773,Z 334.41,A -85,B 0,C 180,E1 23254.829,E2 23254.829} C_VEL
LIN {X 0,Y 640.755,Z 334.404,A -85,B 0,C 180,E1 23251.728,E2 23251.728} C_VEL
LIN {X 0,Y 640.737,Z 334.412,A -85,B 0,C 180,E1 23249.136,E2 23249.136} C_VEL
LIN {X 0,Y 640.815,Z 334.381,A -85,B 0,C 180,E1 23246.205,E2 23246.205} C_VEL
LIN {X 0,Y 640.731,Z 334.412,A -85,B 0,C 180,E1 23243.2,E2 23243.2} C_VEL
LIN {X 0,Y 640.741,Z 334.397,A -85,B 0,C 180,E1 23240.651,E2 23240.651} C_VEL
LIN {X 0,Y 640.744,Z 334.393,A -85,B 0,C 180,E1 23237.435,E2 23237.435} C_VEL
LIN {X 0,Y 640.722,Z 334.412,A -85,B 0,C 180,E1 23234.829,E2 23234.829} C_VEL
LIN {X 0,Y 640.8,Z 334.384,A -85,B 0,C 180,E1 23231.949,E2 23231.949} C_VEL
LIN {X 0,Y 640.728,Z 334.415,A -85,B 0,C 180,E1 23228.957,E2 23228.957} C_VEL
LIN {X 0,Y 640.734,Z 334.394,A -85,B 0,C 180,E1 23226.451,E2 23226.451} C_VEL
LIN {X 0,Y 640.791,Z 334.413,A -85,B 0,C 180,E1 23223.399,E2 23223.399} C_VEL
LIN {X 0,Y 640.733,Z 334.387,A -85,B 0,C 180,E1 23220.626,E2 23220.626} C_VEL
LIN {X 0,Y 640.772,Z 334.41,A -85,B 0,C 180,E1 23217.943,E2 23217.943} C_VEL
LIN {X 0,Y 640.75,Z 334.383,A -85,B 0,C 180,E1 23214.807,E2 23214.807} C_VEL
LIN {X 0,Y 640.75,Z 334.413,A -85,B 0,C 180,E1 23212.197,E2 23212.197} C_VEL
LIN {X 0,Y 640.808,Z 334.382,A -85,B 0,C 180,E1 23209.117,E2 23209.117} C_VEL
LIN {X 0,Y 640.752,Z 334.411,A -85,B 0,C 180,E1 23206.279,E2 23206.279} C_VEL
LIN {X 0,Y 640.796,Z 334.384,A -85,B 0,C 180,E1 23203.501,E2 23203.501} C_VEL
LIN {X 0,Y 640.763,Z 334.394,A -85,B 0,C 180,E1 23200.397,E2 23200.397} C_VEL
LIN {X 0,Y 640.768,Z 334.411,A -85,B 0,C 180,E1 23197.716,E2 23197.716} C_VEL
LIN {X 0,Y 640.799,Z 334.39,A -85,B 0,C 180,E1 23194.589,E2 23194.589} C_VEL
LIN {X 0,Y 640.766,Z 334.41,A -85,B 0,C 180,E1 23191.782,E2 23191.782} C_VEL
LIN {X 0,Y 640.835,Z 334.405,A -85,B 0,C 180,E1 23188.762,E2 23188.762} C_VEL
LIN {X 0,Y 640.79,Z 334.536,A -85,B 0,C 180,E1 23187.582,E2 23187.582} C_VEL
LIN {X 0,Y 642.196,Z 338.003,A -85,B 0,C 180,E1 23187.085,E2 23187.085} C_VEL
LIN {X 0,Y 643.142,Z 339.66,A -85,B 0,C 180,E1 23186.821,E2 23186.821} C_VEL
LIN {X 0,Y 644.311,Z 342.118,A -85,B 0,C 180,E1 23186.517,E2 23186.517} C_VEL
LIN {X 0,Y 653.876,Z 355.119,A -85,B 0,C 180,E1 23185.29,E2 23185.29} C_VEL
LIN {X 0,Y 665.984,Z 372.484,A -85,B 0,C 180,E1 23183.813,E2 23183.813} C_VEL
LIN {X 0,Y 672.604,Z 382.646,A -85,B 0,C 180,E1 23183.036,E2 23183.036} C_VEL
LIN {X 0,Y 671.657,Z 434.517,A -85,B 0,C 180,E1 23182.33,E2 23182.33} C_VEL
LIN {X 0,Y 670.845,Z 442.219,A -85,B 0,C 180,E1 23182.286,E2 23182.286} C_VEL
LIN {X 0,Y 666.137,Z 462.903,A -85,B 0,C 180,E1 23182.394,E2 23182.394} C_VEL
LIN {X 0,Y 665.458,Z 469.518,A -85,B 0,C 180,E1 23182.354,E2 23182.354} C_VEL
LIN {X 0,Y 661.552,Z 683.299,A -85,B 0,C 180,E1 23179.487,E2 23179.487} C_VEL
LIN {X 0,Y 659.077,Z 817.87,A -85,B 0,C 180,E1 23177.703,E2 23177.703} C_VEL
LIN {X 0,Y 658.113,Z 842.922,A -85,B 0,C 180,E1 23177.254,E2 23177.254} C_VEL
LIN {X 0,Y 656.621,Z 870.799,A -85,B 0,C 180,E1 23176.573,E2 23176.573} C_VEL
LIN {X 0,Y 655.228,Z 892.555,A -85,B 0,C 180,E1 23175.903,E2 23175.903} C_VEL
LIN {X 0,Y 653.838,Z 912.087,A -85,B 0,C 180,E1 23175.199,E2 23175.199} C_VEL
LIN {X 0,Y 652.223,Z 932.508,A -85,B 0,C 180,E1 23174.351,E2 23174.351} C_VEL
LIN {X 0,Y 650.418,Z 954.06,A -85,B 0,C 180,E1 23173.323,E2 23173.323} C_VEL
LIN {X 0,Y 648.123,Z 979.585,A -85,B 0,C 180,E1 23171.912,E2 23171.912} C_VEL
LIN {X 0,Y 646.127,Z 1000.312,A -85,B 0,C 180,E1 23170.595,E2 23170.595} C_VEL
LIN {X 0,Y 644.317,Z 1018.822,A -85,B 0,C 180,E1 23169.282,E2 23169.282} C_VEL
LIN {X 0,Y 642.423,Z 1038.227,A -85,B 0,C 180,E1 23167.751,E2 23167.751} C_VEL
LIN {X 0,Y 640.32,Z 1060.194,A -85,B 0,C 180,E1 23165.788,E2 23165.788} C_VEL
LIN {X 0,Y 638.729,Z 1077.153,A -85,B 0,C 180,E1 23164.084,E2 23164.084} C_VEL
LIN {X 0,Y 637.168,Z 1094.596,A -85,B 0,C 180,E1 23162.139,E2 23162.139} C_VEL
LIN {X 0,Y 635.724,Z 1112.208,A -85,B 0,C 180,E1 23159.906,E2 23159.906} C_VEL
LIN {X 0,Y 634.733,Z 1125.602,A -85,B 0,C 180,E1 23157.997,E2 23157.997} C_VEL
LIN {X 0,Y 633.805,Z 1139.873,A -85,B 0,C 180,E1 23155.711,E2 23155.711} C_VEL
LIN {X 0,Y 633.077,Z 1152.532,A -85,B 0,C 180,E1 23153.355,E2 23153.355} C_VEL
LIN {X 0,Y 632.63,Z 1162.066,A -85,B 0,C 180,E1 23151.316,E2 23151.316} C_VEL
LIN {X 0,Y 632.322,Z 1170.393,A -85,B 0,C 180,E1 23149.258,E2 23149.258} C_VEL
LIN {X 0,Y 632.106,Z 1178.401,A -85,B 0,C 180,E1 23146.921,E2 23146.921} C_VEL
LIN {X 0,Y 631.991,Z 1184.991,A -85,B 0,C 180,E1 23144.473,E2 23144.473} C_VEL
LIN {X 0,Y 631.933,Z 1189.529,A -85,B 0,C 180,E1 23142.24,E2 23142.24} C_VEL
LIN {X 0,Y 631.911,Z 1192.806,A -85,B 0,C 180,E1 23139.931,E2 23139.931} C_VEL
LIN {X 0,Y 631.91,Z 1194.611,A -85,B 0,C 180,E1 23137.546,E2 23137.546} C_VEL
LIN {X 0,Y 631.899,Z 1194.858,A -85,B 0,C 180,E1 23135.356,E2 23135.356} C_VEL
LIN {X 0,Y 631.91,Z 1193.962,A -85,B 0,C 180,E1 23133.265,E2 23133.265} C_VEL
LIN {X 0,Y 631.921,Z 1191.601,A -85,B 0,C 180,E1 23130.997,E2 23130.997} C_VEL
LIN {X 0,Y 631.953,Z 1187.45,A -85,B 0,C 180,E1 23128.549,E2 23128.549} C_VEL
LIN {X 0,Y 632.033,Z 1181.82,A -85,B 0,C 180,E1 23126.19,E2 23126.19} C_VEL
LIN {X 0,Y 632.193,Z 1174.933,A -85,B 0,C 180,E1 23123.917,E2 23123.917} C_VEL
LIN {X 0,Y 632.52,Z 1165.394,A -85,B 0,C 180,E1 23121.363,E2 23121.363} C_VEL
LIN {X 0,Y 632.956,Z 1155.072,A -85,B 0,C 180,E1 23119.072,E2 23119.072} C_VEL
LIN {X 0,Y 633.507,Z 1144.606,A -85,B 0,C 180,E1 23117.048,E2 23117.048} C_VEL
LIN {X 0,Y 634.312,Z 1131.582,A -85,B 0,C 180,E1 23114.831,E2 23114.831} C_VEL
LIN {X 0,Y 635.446,Z 1115.617,A -85,B 0,C 180,E1 23112.47,E2 23112.47} C_VEL
LIN {X 0,Y 636.648,Z 1100.971,A -85,B 0,C 180,E1 23110.552,E2 23110.552} C_VEL
LIN {X 0,Y 638.228,Z 1082.566,A -85,B 0,C 180,E1 23108.397,E2 23108.397} C_VEL
LIN {X 0,Y 639.921,Z 1064.292,A -85,B 0,C 180,E1 23106.519,E2 23106.519} C_VEL
LIN {X 0,Y 641.513,Z 1047.549,A -85,B 0,C 180,E1 23104.965,E2 23104.965} C_VEL
LIN {X 0,Y 643.399,Z 1028.441,A -85,B 0,C 180,E1 23103.362,E2 23103.362} C_VEL
LIN {X 0,Y 645.613,Z 1005.445,A -85,B 0,C 180,E1 23101.661,E2 23101.661} C_VEL
LIN {X 0,Y 647.486,Z 985.935,A -85,B 0,C 180,E1 23100.385,E2 23100.385} C_VEL
LIN {X 0,Y 649.328,Z 966.2,A -85,B 0,C 180,E1 23099.234,E2 23099.234} C_VEL
LIN {X 0,Y 651.355,Z 943.68,A -85,B 0,C 180,E1 23098.073,E2 23098.073} C_VEL
LIN {X 0,Y 653.437,Z 917.903,A -85,B 0,C 180,E1 23096.94,E2 23096.94} C_VEL
LIN {X 0,Y 654.948,Z 896.397,A -85,B 0,C 180,E1 23096.135,E2 23096.135} C_VEL
LIN {X 0,Y 656.391,Z 874.451,A -85,B 0,C 180,E1 23095.442,E2 23095.442} C_VEL
LIN {X 0,Y 657.74,Z 850.366,A -85,B 0,C 180,E1 23094.82,E2 23094.82} C_VEL
LIN {X 0,Y 658.966,Z 821.688,A -85,B 0,C 180,E1 23094.265,E2 23094.265} C_VEL
LIN {X 0,Y 659.982,Z 774.341,A -85,B 0,C 180,E1 23093.621,E2 23093.621} C_VEL
LIN {X 0,Y 663.908,Z 552.206,A -85,B 0,C 180,E1 23090.675,E2 23090.675} C_VEL
LIN {X 0,Y 666.986,Z 386.072,A -85,B 0,C 180,E1 23088.405,E2 23088.405} C_VEL
LIN {X 0,Y 654.65,Z 367.843,A -85,B 0,C 180,E1 23086.91,E2 23086.91} C_VEL
LIN {X 0,Y 644.268,Z 353.333,A -85,B 0,C 180,E1 23085.583,E2 23085.583} C_VEL
LIN {X 0,Y 636.883,Z 343.518,A -85,B 0,C 180,E1 23084.602,E2 23084.602} C_VEL
LIN {X 0,Y 635.272,Z 340.919,A -85,B 0,C 180,E1 23084.334,E2 23084.334} C_VEL
LIN {X 0,Y 633.068,Z 336.344,A -85,B 0,C 180,E1 23083.647,E2 23083.647} C_VEL
LIN {X 0,Y 632.889,Z 335.391,A -85,B 0,C 180,E1 23083.518,E2 23083.518} C_VEL
LIN {X 0,Y 632.861,Z 335.401,A -85,B 0,C 180,E1 23080.375,E2 23080.375} C_VEL
LIN {X 0,Y 632.892,Z 335.391,A -85,B 0,C 180,E1 23077.35,E2 23077.35} C_VEL
LIN {X 0,Y 632.855,Z 335.4,A -85,B 0,C 180,E1 23074.227,E2 23074.227} C_VEL
LIN {X 0,Y 632.894,Z 335.394,A -85,B 0,C 180,E1 23071.212,E2 23071.212} C_VEL
LIN {X 0,Y 632.849,Z 335.388,A -85,B 0,C 180,E1 23068.162,E2 23068.162} C_VEL
LIN {X 0,Y 632.888,Z 335.373,A -85,B 0,C 180,E1 23065.141,E2 23065.141} C_VEL
LIN {X 0,Y 632.846,Z 335.386,A -85,B 0,C 180,E1 23062.089,E2 23062.089} C_VEL
LIN {X 0,Y 632.879,Z 335.37,A -85,B 0,C 180,E1 23059.089,E2 23059.089} C_VEL
LIN {X 0,Y 632.838,Z 335.39,A -85,B 0,C 180,E1 23055.957,E2 23055.957} C_VEL
LIN {X 0,Y 632.861,Z 335.358,A -85,B 0,C 180,E1 23053.058,E2 23053.058} C_VEL
LIN {X 0,Y 632.839,Z 335.398,A -85,B 0,C 180,E1 23049.917,E2 23049.917} C_VEL
LIN {X 0,Y 632.841,Z 335.397,A -85,B 0,C 180,E1 23047.079,E2 23047.079} C_VEL
LIN {X 0,Y 632.831,Z 335.402,A -85,B 0,C 180,E1 23043.805,E2 23043.805} C_VEL
LIN {X 0,Y 632.825,Z 335.392,A -85,B 0,C 180,E1 23041.086,E2 23041.086} C_VEL
LIN {X 0,Y 632.848,Z 335.393,A -85,B 0,C 180,E1 23037.917,E2 23037.917} C_VEL
LIN {X 0,Y 632.811,Z 335.396,A -85,B 0,C 180,E1 23035.105,E2 23035.105} C_VEL
LIN {X 0,Y 632.884,Z 335.392,A -85,B 0,C 180,E1 23032.1,E2 23032.1} C_VEL
LIN {X 0,Y 632.801,Z 335.402,A -85,B 0,C 180,E1 23029.162,E2 23029.162} C_VEL
LIN {X 0,Y 632.852,Z 335.361,A -85,B 0,C 180,E1 23026.291,E2 23026.291} C_VEL
LIN {X 0,Y 632.799,Z 335.404,A -85,B 0,C 180,E1 23023.243,E2 23023.243} C_VEL
LIN {X 0,Y 632.804,Z 335.369,A -85,B 0,C 180,E1 23020.525,E2 23020.525} C_VEL
LIN {X 0,Y 632.809,Z 335.403,A -85,B 0,C 180,E1 23017.323,E2 23017.323} C_VEL
LIN {X 0,Y 632.784,Z 335.368,A -85,B 0,C 180,E1 23014.645,E2 23014.645} C_VEL
LIN {X 0,Y 632.864,Z 335.394,A -85,B 0,C 180,E1 23011.604,E2 23011.604} C_VEL
LIN {X 0,Y 632.793,Z 335.398,A -85,B 0,C 180,E1 23008.742,E2 23008.742} C_VEL
LIN {X 0,Y 632.837,Z 335.403,A -85,B 0,C 180,E1 23005.991,E2 23005.991} C_VEL
LIN {X 0,Y 632.87,Z 335.615,A -85,B 0,C 180,E1 23003.179,E2 23003.179} C_VEL
LIN {X 0,Y 634.102,Z 338.877,A -85,B 0,C 180,E1 23002.734,E2 23002.734} C_VEL
LIN {X 0,Y 635.116,Z 340.564,A -85,B 0,C 180,E1 23002.463,E2 23002.463} C_VEL
LIN {X 0,Y 639.608,Z 349.771,A -85,B 0,C 180,E1 23001.124,E2 23001.124} C_VEL
LIN {X 0,Y 650.044,Z 364.519,A -85,B 0,C 180,E1 22999.727,E2 22999.727} C_VEL
LIN {X 0,Y 662.367,Z 382.289,A -85,B 0,C 180,E1 22998.204,E2 22998.204} C_VEL
LIN {X 0,Y 667.17,Z 389.702,A -85,B 0,C 180,E1 22997.63,E2 22997.63} C_VEL
LIN {X 0,Y 663.27,Z 596.963,A -85,B 0,C 180,E1 22994.814,E2 22994.814} C_VEL
LIN {X 0,Y 659.343,Z 819.382,A -85,B 0,C 180,E1 22991.872,E2 22991.872} C_VEL
LIN {X 0,Y 658.475,Z 843.898,A -85,B 0,C 180,E1 22991.475,E2 22991.475} C_VEL
LIN {X 0,Y 657.4,Z 866.761,A -85,B 0,C 180,E1 22990.982,E2 22990.982} C_VEL
LIN {X 0,Y 655.941,Z 892.478,A -85,B 0,C 180,E1 22990.279,E2 22990.279} C_VEL
LIN {X 0,Y 654.085,Z 918.716,A -85,B 0,C 180,E1 22989.375,E2 22989.375} C_VEL
LIN {X 0,Y 652.376,Z 940.583,A -85,B 0,C 180,E1 22988.482,E2 22988.482} C_VEL
LIN {X 0,Y 650.529,Z 962.704,A -85,B 0,C 180,E1 22987.437,E2 22987.437} C_VEL
LIN {X 0,Y 648.186,Z 988.943,A -85,B 0,C 180,E1 22985.996,E2 22985.996} C_VEL
LIN {X 0,Y 646.23,Z 1009.32,A -85,B 0,C 180,E1 22984.708,E2 22984.708} C_VEL
LIN {X 0,Y 644.435,Z 1027.72,A -85,B 0,C 180,E1 22983.41,E2 22983.41} C_VEL
LIN {X 0,Y 642.597,Z 1046.473,A -85,B 0,C 180,E1 22981.941,E2 22981.941} C_VEL
LIN {X 0,Y 640.406,Z 1069.078,A -85,B 0,C 180,E1 22979.94,E2 22979.94} C_VEL
LIN {X 0,Y 638.846,Z 1085.914,A -85,B 0,C 180,E1 22978.259,E2 22978.259} C_VEL
LIN {X 0,Y 637.369,Z 1102.221,A -85,B 0,C 180,E1 22976.457,E2 22976.457} C_VEL
LIN {X 0,Y 635.893,Z 1120.245,A -85,B 0,C 180,E1 22974.216,E2 22974.216} C_VEL
LIN {X 0,Y 634.769,Z 1134.906,A -85,B 0,C 180,E1 22972.146,E2 22972.146} C_VEL
LIN {X 0,Y 633.906,Z 1147.728,A -85,B 0,C 180,E1 22970.112,E2 22970.112} C_VEL
LIN {X 0,Y 633.147,Z 1161.283,A -85,B 0,C 180,E1 22967.651,E2 22967.651} C_VEL
LIN {X 0,Y 632.66,Z 1171.077,A -85,B 0,C 180,E1 22965.586,E2 22965.586} C_VEL
LIN {X 0,Y 632.373,Z 1179.157,A -85,B 0,C 180,E1 22963.627,E2 22963.627} C_VEL
LIN {X 0,Y 632.15,Z 1186.708,A -85,B 0,C 180,E1 22961.496,E2 22961.496} C_VEL
LIN {X 0,Y 632.004,Z 1193.594,A -85,B 0,C 180,E1 22959.103,E2 22959.103} C_VEL
LIN {X 0,Y 631.939,Z 1198.921,A -85,B 0,C 180,E1 22956.633,E2 22956.633} C_VEL
LIN {X 0,Y 631.917,Z 1202.356,A -85,B 0,C 180,E1 22954.356,E2 22954.356} C_VEL
LIN {X 0,Y 631.911,Z 1204.438,A -85,B 0,C 180,E1 22951.995,E2 22951.995} C_VEL
LIN {X 0,Y 631.892,Z 1204.894,A -85,B 0,C 180,E1 22949.547,E2 22949.547} C_VEL
LIN {X 0,Y 631.91,Z 1204.007,A -85,B 0,C 180,E1 22947.37,E2 22947.37} C_VEL
LIN {X 0,Y 631.921,Z 1201.675,A -85,B 0,C 180,E1 22945.099,E2 22945.099} C_VEL
LIN {X 0,Y 631.956,Z 1197.543,A -85,B 0,C 180,E1 22942.637,E2 22942.637} C_VEL
LIN {X 0,Y 632.034,Z 1191.876,A -85,B 0,C 180,E1 22940.255,E2 22940.255} C_VEL
LIN {X 0,Y 632.182,Z 1184.891,A -85,B 0,C 180,E1 22937.95,E2 22937.95} C_VEL
LIN {X 0,Y 632.529,Z 1175.145,A -85,B 0,C 180,E1 22935.35,E2 22935.35} C_VEL
LIN {X 0,Y 632.943,Z 1165,A -85,B 0,C 180,E1 22933.102,E2 22933.102} C_VEL
LIN {X 0,Y 633.497,Z 1154.763,A -85,B 0,C 180,E1 22931.122,E2 22931.122} C_VEL
LIN {X 0,Y 634.299,Z 1141.95,A -85,B 0,C 180,E1 22928.937,E2 22928.937} C_VEL
LIN {X 0,Y 635.434,Z 1125.798,A -85,B 0,C 180,E1 22926.541,E2 22926.541} C_VEL
LIN {X 0,Y 636.63,Z 1111.083,A -85,B 0,C 180,E1 22924.611,E2 22924.611} C_VEL
LIN {X 0,Y 638.207,Z 1092.835,A -85,B 0,C 180,E1 22922.47,E2 22922.47} C_VEL
LIN {X 0,Y 639.968,Z 1073.814,A -85,B 0,C 180,E1 22920.518,E2 22920.518} C_VEL
LIN {X 0,Y 641.533,Z 1057.514,A -85,B 0,C 180,E1 22919.007,E2 22919.007} C_VEL
LIN {X 0,Y 643.32,Z 1039.188,A -85,B 0,C 180,E1 22917.469,E2 22917.469} C_VEL
LIN {X 0,Y 645.643,Z 1015.188,A -85,B 0,C 180,E1 22915.688,E2 22915.688} C_VEL
LIN {X 0,Y 647.617,Z 994.63,A -85,B 0,C 180,E1 22914.35,E2 22914.35} C_VEL
LIN {X 0,Y 649.503,Z 974.414,A -85,B 0,C 180,E1 22913.181,E2 22913.181} C_VEL
LIN {X 0,Y 651.752,Z 949.299,A -85,B 0,C 180,E1 22911.909,E2 22911.909} C_VEL
LIN {X 0,Y 653.674,Z 924.583,A -85,B 0,C 180,E1 22910.854,E2 22910.854} C_VEL
LIN {X 0,Y 655.116,Z 904.124,A -85,B 0,C 180,E1 22910.104,E2 22910.104} C_VEL
LIN {X 0,Y 656.513,Z 882.372,A -85,B 0,C 180,E1 22909.427,E2 22909.427} C_VEL
LIN {X 0,Y 657.913,Z 857.298,A -85,B 0,C 180,E1 22908.795,E2 22908.795} C_VEL
LIN {X 0,Y 659.043,Z 829.264,A -85,B 0,C 180,E1 22908.272,E2 22908.272} C_VEL
LIN {X 0,Y 660.738,Z 740.201,A -85,B 0,C 180,E1 22907.087,E2 22907.087} C_VEL
LIN {X 0,Y 664.742,Z 517.949,A -85,B 0,C 180,E1 22904.124,E2 22904.124} C_VEL
LIN {X 0,Y 667.126,Z 389.324,A -85,B 0,C 180,E1 22902.36,E2 22902.36} C_VEL
LIN {X 0,Y 652.194,Z 367.51,A -85,B 0,C 180,E1 22900.545,E2 22900.545} C_VEL
LIN {X 0,Y 641.849,Z 353.061,A -85,B 0,C 180,E1 22899.205,E2 22899.205} C_VEL
LIN {X 0,Y 639.642,Z 349.809,A -85,B 0,C 180,E1 22898.881,E2 22898.881} C_VEL
LIN {X 0,Y 636.764,Z 343.845,A -85,B 0,C 180,E1 22897.992,E2 22897.992} C_VEL
LIN {X 0,Y 634.693,Z 339.646,A -85,B 0,C 180,E1 22897.339,E2 22897.339} C_VEL
LIN {X 0,Y 633.163,Z 336.871,A -85,B 0,C 180,E1 22896.877,E2 22896.877} C_VEL
LIN {X 0,Y 632.862,Z 335.397,A -85,B 0,C 180,E1 22896.671,E2 22896.671} C_VEL
LIN {X 0,Y 632.807,Z 335.4,A -85,B 0,C 180,E1 22893.575,E2 22893.575} C_VEL
LIN {X 0,Y 632.813,Z 335.378,A -85,B 0,C 180,E1 22890.899,E2 22890.899} C_VEL
LIN {X 0,Y 632.817,Z 335.394,A -85,B 0,C 180,E1 22887.681,E2 22887.681} C_VEL
LIN {X 0,Y 632.799,Z 335.397,A -85,B 0,C 180,E1 22884.954,E2 22884.954} C_VEL
LIN {X 0,Y 632.854,Z 335.37,A -85,B 0,C 180,E1 22881.893,E2 22881.893} C_VEL
LIN {X 0,Y 632.789,Z 335.405,A -85,B 0,C 180,E1 22878.996,E2 22878.996} C_VEL
LIN {X 0,Y 632.859,Z 335.369,A -85,B 0,C 180,E1 22876.051,E2 22876.051} C_VEL
LIN {X 0,Y 632.789,Z 335.4,A -85,B 0,C 180,E1 22873.059,E2 22873.059} C_VEL
LIN {X 0,Y 632.804,Z 335.381,A -85,B 0,C 180,E1 22870.377,E2 22870.377} C_VEL
LIN {X 0,Y 632.805,Z 335.389,A -85,B 0,C 180,E1 22867.127,E2 22867.127} C_VEL
LIN {X 0,Y 632.799,Z 335.391,A -85,B 0,C 180,E1 22864.421,E2 22864.421} C_VEL
LIN {X 0,Y 632.852,Z 335.376,A -85,B 0,C 180,E1 22861.358,E2 22861.358} C_VEL
LIN {X 0,Y 632.799,Z 335.398,A -85,B 0,C 180,E1 22858.551,E2 22858.551} C_VEL
LIN {X 0,Y 632.863,Z 335.372,A -85,B 0,C 180,E1 22855.651,E2 22855.651} C_VEL
LIN {X 0,Y 632.813,Z 335.402,A -85,B 0,C 180,E1 22852.647,E2 22852.647} C_VEL
LIN {X 0,Y 632.816,Z 335.378,A -85,B 0,C 180,E1 22849.991,E2 22849.991} C_VEL
LIN {X 0,Y 632.835,Z 335.399,A -85,B 0,C 180,E1 22846.722,E2 22846.722} C_VEL
LIN {X 0,Y 632.813,Z 335.369,A -85,B 0,C 180,E1 22844.042,E2 22844.042} C_VEL
LIN {X 0,Y 632.887,Z 335.383,A -85,B 0,C 180,E1 22841.007,E2 22841.007} C_VEL
LIN {X 0,Y 632.819,Z 335.399,A -85,B 0,C 180,E1 22838.044,E2 22838.044} C_VEL
LIN {X 0,Y 632.889,Z 335.368,A -85,B 0,C 180,E1 22835.071,E2 22835.071} C_VEL
LIN {X 0,Y 632.825,Z 335.398,A -85,B 0,C 180,E1 22832.013,E2 22832.013} C_VEL
LIN {X 0,Y 632.88,Z 335.395,A -85,B 0,C 180,E1 22829.105,E2 22829.105} C_VEL
LIN {X 0,Y 632.882,Z 335.509,A -85,B 0,C 180,E1 22828.447,E2 22828.447} C_VEL
LIN {X 0,Y 633.972,Z 338.628,A -85,B 0,C 180,E1 22827.999,E2 22827.999} C_VEL
LIN {X 0,Y 635.224,Z 340.687,A -85,B 0,C 180,E1 22827.643,E2 22827.643} C_VEL
LIN {X 0,Y 636.159,Z 342.544,A -85,B 0,C 180,E1 22827.43,E2 22827.43} C_VEL
LIN {X 0,Y 642.254,Z 350.549,A -85,B 0,C 180,E1 22826.596,E2 22826.596} C_VEL
LIN {X 0,Y 653.49,Z 366.186,A -85,B 0,C 180,E1 22825.146,E2 22825.146} C_VEL
LIN {X 0,Y 665.374,Z 383.68,A -85,B 0,C 180,E1 22823.695,E2 22823.695} C_VEL
LIN {X 0,Y 667.08,Z 386.52,A -85,B 0,C 180,E1 22823.489,E2 22823.489} C_VEL
LIN {X 0,Y 665.458,Z 469.518,A -85,B 0,C 180,E1 22822.354,E2 22822.354} C_VEL
LIN {X 0,Y 664.581,Z 477.227,A -85,B 0,C 180,E1 22822.315,E2 22822.315} C_VEL
LIN {X 0,Y 659.845,Z 497.897,A -85,B 0,C 180,E1 22822.427,E2 22822.427} C_VEL
LIN {X 0,Y 659.206,Z 504.502,A -85,B 0,C 180,E1 22822.383,E2 22822.383} C_VEL
LIN {X 0,Y 655.206,Z 712.153,A -85,B 0,C 180,E1 22819.587,E2 22819.587} C_VEL
LIN {X 0,Y 653.097,Z 818.022,A -85,B 0,C 180,E1 22818.17,E2 22818.17} C_VEL
LIN {X 0,Y 652.069,Z 843.037,A -85,B 0,C 180,E1 22817.719,E2 22817.719} C_VEL
LIN {X 0,Y 650.491,Z 870.851,A -85,B 0,C 180,E1 22817.036,E2 22817.036} C_VEL
LIN {X 0,Y 648.985,Z 892.949,A -85,B 0,C 180,E1 22816.351,E2 22816.351} C_VEL
LIN {X 0,Y 647.492,Z 912.499,A -85,B 0,C 180,E1 22815.641,E2 22815.641} C_VEL
LIN {X 0,Y 645.722,Z 933.521,A -85,B 0,C 180,E1 22814.758,E2 22814.758} C_VEL
LIN {X 0,Y 643.625,Z 957.166,A -85,B 0,C 180,E1 22813.61,E2 22813.61} C_VEL
LIN {X 0,Y 641.18,Z 981.889,A -85,B 0,C 180,E1 22812.205,E2 22812.205} C_VEL
LIN {X 0,Y 639.27,Z 1000.521,A -85,B 0,C 180,E1 22811.005,E2 22811.005} C_VEL
LIN {X 0,Y 637.414,Z 1018.303,A -85,B 0,C 180,E1 22809.733,E2 22809.733} C_VEL
LIN {X 0,Y 635.517,Z 1036.307,A -85,B 0,C 180,E1 22808.308,E2 22808.308} C_VEL
LIN {X 0,Y 633.302,Z 1057.648,A -85,B 0,C 180,E1 22806.415,E2 22806.415} C_VEL
LIN {X 0,Y 631.447,Z 1075.958,A -85,B 0,C 180,E1 22804.571,E2 22804.571} C_VEL
LIN {X 0,Y 629.886,Z 1092.053,A -85,B 0,C 180,E1 22802.772,E2 22802.772} C_VEL
LIN {X 0,Y 628.271,Z 1110.075,A -85,B 0,C 180,E1 22800.509,E2 22800.509} C_VEL
LIN {X 0,Y 627.044,Z 1125.027,A -85,B 0,C 180,E1 22798.371,E2 22798.371} C_VEL
LIN {X 0,Y 626.076,Z 1138.166,A -85,B 0,C 180,E1 22796.256,E2 22796.256} C_VEL
LIN {X 0,Y 625.24,Z 1151.637,A -85,B 0,C 180,E1 22793.765,E2 22793.765} C_VEL
LIN {X 0,Y 624.717,Z 1161.705,A -85,B 0,C 180,E1 22791.599,E2 22791.599} C_VEL
LIN {X 0,Y 624.389,Z 1169.571,A -85,B 0,C 180,E1 22789.65,E2 22789.65} C_VEL
LIN {X 0,Y 624.173,Z 1176.939,A -85,B 0,C 180,E1 22787.527,E2 22787.527} C_VEL
LIN {X 0,Y 624.008,Z 1183.907,A -85,B 0,C 180,E1 22785.045,E2 22785.045} C_VEL
LIN {X 0,Y 623.94,Z 1189.067,A -85,B 0,C 180,E1 22782.588,E2 22782.588} C_VEL
LIN {X 0,Y 623.918,Z 1192.386,A -85,B 0,C 180,E1 22780.34,E2 22780.34} C_VEL
LIN {X 0,Y 623.91,Z 1194.47,A -85,B 0,C 180,E1 22777.922,E2 22777.922} C_VEL
LIN {X 0,Y 623.896,Z 1194.877,A -85,B 0,C 180,E1 22775.425,E2 22775.425} C_VEL
LIN {X 0,Y 623.909,Z 1194.016,A -85,B 0,C 180,E1 22773.307,E2 22773.307} C_VEL
LIN {X 0,Y 623.921,Z 1191.697,A -85,B 0,C 180,E1 22771.01,E2 22771.01} C_VEL
LIN {X 0,Y 623.955,Z 1187.612,A -85,B 0,C 180,E1 22768.53,E2 22768.53} C_VEL
LIN {X 0,Y 624.042,Z 1182.027,A -85,B 0,C 180,E1 22766.141,E2 22766.141} C_VEL
LIN {X 0,Y 624.214,Z 1175.181,A -85,B 0,C 180,E1 22763.839,E2 22763.839} C_VEL
LIN {X 0,Y 624.551,Z 1166.103,A -85,B 0,C 180,E1 22761.344,E2 22761.344} C_VEL
LIN {X 0,Y 625.035,Z 1155.453,A -85,B 0,C 180,E1 22758.932,E2 22758.932} C_VEL
LIN {X 0,Y 625.64,Z 1145.045,A -85,B 0,C 180,E1 22756.883,E2 22756.883} C_VEL
LIN {X 0,Y 626.458,Z 1132.639,A -85,B 0,C 180,E1 22754.731,E2 22754.731} C_VEL
LIN {X 0,Y 627.649,Z 1117.157,A -85,B 0,C 180,E1 22752.381,E2 22752.381} C_VEL
LIN {X 0,Y 628.947,Z 1102.363,A -85,B 0,C 180,E1 22750.4,E2 22750.4} C_VEL
LIN {X 0,Y 630.461,Z 1085.802,A -85,B 0,C 180,E1 22748.411,E2 22748.411} C_VEL
LIN {X 0,Y 632.438,Z 1066.105,A -85,B 0,C 180,E1 22746.323,E2 22746.323} C_VEL
LIN {X 0,Y 634.18,Z 1049.001,A -85,B 0,C 180,E1 22744.705,E2 22744.705} C_VEL
LIN {X 0,Y 635.964,Z 1032.111,A -85,B 0,C 180,E1 22743.258,E2 22743.258} C_VEL
LIN {X 0,Y 638.035,Z 1012.385,A -85,B 0,C 180,E1 22741.731,E2 22741.731} C_VEL
LIN {X 0,Y 640.464,Z 988.796,A -85,B 0,C 180,E1 22740.131,E2 22740.131} C_VEL
LIN {X 0,Y 642.454,Z 968.845,A -85,B 0,C 180,E1 22738.94,E2 22738.94} C_VEL
LIN {X 0,Y 644.331,Z 949.109,A -85,B 0,C 180,E1 22737.893,E2 22737.893} C_VEL
LIN {X 0,Y 646.245,Z 927.732,A -85,B 0,C 180,E1 22736.895,E2 22736.895} C_VEL
LIN {X 0,Y 648.463,Z 900.133,A -85,B 0,C 180,E1 22735.804,E2 22735.804} C_VEL
LIN {X 0,Y 650.121,Z 876.462,A -85,B 0,C 180,E1 22735.037,E2 22735.037} C_VEL
LIN {X 0,Y 651.452,Z 854.278,A -85,B 0,C 180,E1 22734.447,E2 22734.447} C_VEL
LIN {X 0,Y 652.715,Z 828.791,A -85,B 0,C 180,E1 22733.913,E2 22733.913} C_VEL
LIN {X 0,Y 653.707,Z 794.328,A -85,B 0,C 180,E1 22733.41,E2 22733.41} C_VEL
LIN {X 0,Y 657.968,Z 568.194,A -85,B 0,C 180,E1 22730.395,E2 22730.395} C_VEL
LIN {X 0,Y 661.54,Z 390.002,A -85,B 0,C 180,E1 22727.949,E2 22727.949} C_VEL
LIN {X 0,Y 648.311,Z 370.38,A -85,B 0,C 180,E1 22726.301,E2 22726.301} C_VEL
LIN {X 0,Y 636.156,Z 353.605,A -85,B 0,C 180,E1 22724.698,E2 22724.698} C_VEL
LIN {X 0,Y 629.506,Z 344.943,A -85,B 0,C 180,E1 22723.8,E2 22723.8} C_VEL
LIN {X 0,Y 627.225,Z 341.434,A -85,B 0,C 180,E1 22723.462,E2 22723.462} C_VEL
LIN {X 0,Y 625.139,Z 337.405,A -85,B 0,C 180,E1 22722.826,E2 22722.826} C_VEL
LIN {X 0,Y 624.937,Z 336.385,A -85,B 0,C 180,E1 22722.688,E2 22722.688} C_VEL
LIN {X 0,Y 624.956,Z 336.387,A -85,B 0,C 180,E1 22719.542,E2 22719.542} C_VEL
LIN {X 0,Y 624.922,Z 336.389,A -85,B 0,C 180,E1 22716.409,E2 22716.409} C_VEL
LIN {X 0,Y 624.954,Z 336.379,A -85,B 0,C 180,E1 22713.284,E2 22713.284} C_VEL
LIN {X 0,Y 624.909,Z 336.386,A -85,B 0,C 180,E1 22710.16,E2 22710.16} C_VEL
LIN {X 0,Y 624.952,Z 336.35,A -85,B 0,C 180,E1 22707.129,E2 22707.129} C_VEL
LIN {X 0,Y 624.905,Z 336.389,A -85,B 0,C 180,E1 22703.98,E2 22703.98} C_VEL
LIN {X 0,Y 624.954,Z 336.347,A -85,B 0,C 180,E1 22701.001,E2 22701.001} C_VEL
LIN {X 0,Y 624.9,Z 336.388,A -85,B 0,C 180,E1 22697.892,E2 22697.892} C_VEL
LIN {X 0,Y 624.947,Z 336.353,A -85,B 0,C 180,E1 22694.903,E2 22694.903} C_VEL
LIN {X 0,Y 624.893,Z 336.378,A -85,B 0,C 180,E1 22691.819,E2 22691.819} C_VEL
LIN {X 0,Y 624.926,Z 336.381,A -85,B 0,C 180,E1 22688.929,E2 22688.929} C_VEL
